LIN {X 0.160,Y -535.997,Z 395.131,A 0.000,B 0.000,C 90.000,E1 59.537} C_DIS
LIN {X 0.035,Y -538.957,Z 395.125,A 0.000,B 0.000,C 90.000,E1 58.408} C_DIS
LIN {X -0.234,Y -540.877,Z 395.120,A 0.000,B 0.000,C 90.000,E1 57.582} C_DIS
LIN {X -0.026,Y -542.349,Z 395.115,A 0.000,B 0.000,C 90.000,E1 56.707} C_DIS
LIN {X 0.021,Y -543.150,Z 395.112,A 0.000,B 0.000,C 90.000,E1 56.135} C_DIS
LIN {X -0.198,Y -544.070,Z 395.107,A 0.000,B 0.000,C 90.000,E1 55.308} C_DIS
LIN {X 0.313,Y -544.582,Z 395.104,A 0.000,B 0.000,C 90.000,E1 54.689} C_DIS
LIN {X 0.100,Y -544.932,Z 395.099,A 0.000,B 0.000,C 90.000,E1 53.863} C_DIS
LIN {X -0.151,Y -544.718,Z 395.091,A 0.000,B 0.000,C 90.000,E1 52.477} C_DIS
LIN {X -0.114,Y -544.668,Z 395.090,A 0.000,B 0.000,C 90.000,E1 52.190} C_DIS
LIN {X 0.024,Y -543.876,Z 395.084,A 0.000,B 0.000,C 90.000,E1 51.045} C_DIS
LIN {X 0.069,Y -542.657,Z 395.077,A 0.000,B 0.000,C 90.000,E1 49.908} C_DIS
LIN {X 0.102,Y -541.174,Z 395.071,A 0.000,B 0.000,C 90.000,E1 48.771} C_DIS
LIN {X -0.280,Y -539.163,Z 395.063,A 0.000,B 0.000,C 90.000,E1 47.391} C_DIS
LIN {X -0.056,Y -534.854,Z 395.047,A 0.000,B 0.000,C 90.000,E1 44.514} C_DIS
LIN {X 0.086,Y -531.734,Z 395.035,A 0.000,B 0.000,C 90.000,E1 42.204} C_DIS
LIN {X -0.062,Y -529.904,Z 395.027,A 0.000,B 0.000,C 90.000,E1 40.782} C_DIS
LIN {X -0.235,Y -528.110,Z 395.019,A 0.000,B 0.000,C 90.000,E1 39.358} C_DIS
LIN {X -0.060,Y -525.925,Z 395.009,A 0.000,B 0.000,C 90.000,E1 37.604} C_DIS
LIN {X 0.091,Y -524.030,Z 395.001,A 0.000,B 0.000,C 90.000,E1 36.137} C_DIS
LIN {X -0.034,Y -521.746,Z 394.991,A 0.000,B 0.000,C 90.000,E1 34.405} C_DIS
LIN {X -0.205,Y -519.458,Z 394.981,A 0.000,B 0.000,C 90.000,E1 32.673} C_DIS
LIN {X 0.171,Y -517.029,Z 394.972,A 0.000,B 0.000,C 90.000,E1 30.875} C_DIS
LIN {X 0.045,Y -514.873,Z 394.962,A 0.000,B 0.000,C 90.000,E1 29.127} C_DIS
LIN {X 0.264,Y -511.965,Z 394.949,A 0.000,B 0.000,C 90.000,E1 26.744} C_DIS
LIN {X -0.248,Y -510.001,Z 394.939,A 0.000,B 0.000,C 90.000,E1 25.027} C_DIS
LIN {X 0.226,Y -507.941,Z 394.927,A 0.000,B 0.000,C 90.000,E1 22.898} C_DIS
LIN {X -0.123,Y -506.318,Z 394.917,A 0.000,B 0.000,C 90.000,E1 21.153} C_DIS
LIN {X 0.245,Y -504.976,Z 394.908,A 0.000,B 0.000,C 90.000,E1 19.322} C_DIS
LIN {X -0.138,Y -503.539,Z 394.896,A 0.000,B 0.000,C 90.000,E1 17.275} C_DIS
LIN {X -0.210,Y -502.689,Z 394.888,A 0.000,B 0.000,C 90.000,E1 15.788} C_DIS
LIN {X 0.103,Y -501.504,Z 394.874,A 0.000,B 0.000,C 90.000,E1 13.355} C_DIS
LIN {X -0.150,Y -500.555,Z 394.854,A 0.000,B 0.000,C 90.000,E1 9.782} C_DIS
LIN {X 0.164,Y -500.484,Z 394.843,A 0.000,B 0.000,C 90.000,E1 7.644} C_DIS
LIN {X 0.217,Y -501.064,Z 394.828,A 0.000,B 0.000,C 90.000,E1 4.935} C_DIS
LIN {X -0.235,Y -503.237,Z 394.806,A 0.000,B 0.000,C 90.000,E1 1.088} C_DIS
LIN {X -0.242,Y -507.371,Z 394.784,A 0.000,B 0.000,C 90.000,E1 357.135} C_DIS
LIN {X 0.074,Y -510.722,Z 394.771,A 0.000,B 0.000,C 90.000,E1 354.723} C_DIS
LIN {X 0.122,Y -514.088,Z 394.759,A 0.000,B 0.000,C 90.000,E1 352.648} C_DIS
LIN {X -0.214,Y -519.053,Z 394.745,A 0.000,B 0.000,C 90.000,E1 350.038} C_DIS
LIN {X -0.215,Y -523.522,Z 394.733,A 0.000,B 0.000,C 90.000,E1 347.993} C_DIS
LIN {X 0.016,Y -528.565,Z 394.722,A 0.000,B 0.000,C 90.000,E1 345.936} C_DIS
LIN {X -0.045,Y -533.123,Z 394.712,A 0.000,B 0.000,C 90.000,E1 344.212} C_DIS
LIN {X -0.056,Y -536.981,Z 394.704,A 0.000,B 0.000,C 90.000,E1 342.779} C_DIS
LIN {X 0.217,Y -541.697,Z 394.695,A 0.000,B 0.000,C 90.000,E1 341.040} C_DIS
LIN {X -0.262,Y -546.551,Z 394.685,A 0.000,B 0.000,C 90.000,E1 339.390} C_DIS
LIN {X -0.168,Y -552.210,Z 394.674,A 0.000,B 0.000,C 90.000,E1 337.411} C_DIS
LIN {X -0.007,Y -556.377,Z 394.667,A 0.000,B 0.000,C 90.000,E1 335.997} C_DIS
LIN {X -0.126,Y -559.734,Z 394.661,A 0.000,B 0.000,C 90.000,E1 334.897} C_DIS
LIN {X 0.193,Y -564.865,Z 394.651,A 0.000,B 0.000,C 90.000,E1 333.204} C_DIS
LIN {X 0.030,Y -569.301,Z 394.644,A 0.000,B 0.000,C 90.000,E1 331.847} C_DIS
LIN {X -0.224,Y -571.851,Z 394.639,A 0.000,B 0.000,C 90.000,E1 331.051} C_DIS
LIN {X 0.218,Y -573.787,Z 394.636,A 0.000,B 0.000,C 90.000,E1 330.461} C_DIS
LIN {X -0.159,Y -579.145,Z 394.627,A 0.000,B 0.000,C 90.000,E1 328.869} C_DIS
LIN {X -0.149,Y -582.761,Z 394.621,A 0.000,B 0.000,C 90.000,E1 327.788} C_DIS
LIN {X -0.046,Y -588.119,Z 394.612,A 0.000,B 0.000,C 90.000,E1 326.167} C_DIS
LIN {X 0.135,Y -592.670,Z 394.605,A 0.000,B 0.000,C 90.000,E1 324.815} C_DIS
LIN {X 0.056,Y -597.283,Z 394.597,A 0.000,B 0.000,C 90.000,E1 323.497} C_DIS
LIN {X -0.047,Y -603.868,Z 394.587,A 0.000,B 0.000,C 90.000,E1 321.662} C_DIS
LIN {X 0.209,Y -609.580,Z 394.578,A 0.000,B 0.000,C 90.000,E1 320.070} C_DIS
LIN {X 0.210,Y -614.342,Z 394.571,A 0.000,B 0.000,C 90.000,E1 318.771} C_DIS
LIN {X 0.295,Y -619.034,Z 394.564,A 0.000,B 0.000,C 90.000,E1 317.472} C_DIS
LIN {X -0.001,Y -623.601,Z 394.557,A 0.000,B 0.000,C 90.000,E1 316.215} C_DIS
LIN {X 0.214,Y -628.170,Z 394.550,A 0.000,B 0.000,C 90.000,E1 314.919} C_DIS
LIN {X -0.147,Y -634.647,Z 394.540,A 0.000,B 0.000,C 90.000,E1 313.176} C_DIS
LIN {X -0.278,Y -640.243,Z 394.531,A 0.000,B 0.000,C 90.000,E1 311.676} C_DIS
LIN {X 0.334,Y -643.911,Z 394.526,A 0.000,B 0.000,C 90.000,E1 310.620} C_DIS
LIN {X 0.089,Y -647.469,Z 394.520,A 0.000,B 0.000,C 90.000,E1 309.644} C_DIS
LIN {X 0.323,Y -651.743,Z 394.513,A 0.000,B 0.000,C 90.000,E1 308.382} C_DIS
LIN {X 0.224,Y -655.835,Z 394.507,A 0.000,B 0.000,C 90.000,E1 307.156} C_DIS
LIN {X 0.187,Y -659.762,Z 394.500,A 0.000,B 0.000,C 90.000,E1 305.931} C_DIS
LIN {X -0.180,Y -663.485,Z 394.493,A 0.000,B 0.000,C 90.000,E1 304.739} C_DIS
LIN {X 0.194,Y -667.864,Z 394.485,A 0.000,B 0.000,C 90.000,E1 303.245} C_DIS
LIN {X -0.054,Y -671.506,Z 394.478,A 0.000,B 0.000,C 90.000,E1 302.054} C_DIS
LIN {X 0.016,Y -674.308,Z 394.473,A 0.000,B 0.000,C 90.000,E1 301.082} C_DIS
LIN {X -0.102,Y -676.921,Z 394.467,A 0.000,B 0.000,C 90.000,E1 300.129} C_DIS
LIN {X 0.057,Y -679.334,Z 394.462,A 0.000,B 0.000,C 90.000,E1 299.155} C_DIS
LIN {X -0.345,Y -681.547,Z 394.457,A 0.000,B 0.000,C 90.000,E1 298.231} C_DIS
LIN {X -0.333,Y -682.891,Z 394.453,A 0.000,B 0.000,C 90.000,E1 297.513} C_DIS
LIN {X -0.125,Y -683.417,Z 394.451,A 0.000,B 0.000,C 90.000,E1 297.257} C_DIS
LIN {X 0.031,Y -685.366,Z 394.445,A 0.000,B 0.000,C 90.000,E1 296.052} C_DIS
LIN {X 0.071,Y -686.370,Z 394.441,A 0.000,B 0.000,C 90.000,E1 295.335} C_DIS
LIN {X -0.176,Y -687.148,Z 394.437,A 0.000,B 0.000,C 90.000,E1 294.643} C_DIS
LIN {X -0.194,Y -687.808,Z 394.432,A 0.000,B 0.000,C 90.000,E1 293.695} C_DIS
LIN {X -0.245,Y -687.936,Z 394.430,A 0.000,B 0.000,C 90.000,E1 293.462} C_DIS
LIN {X -0.038,Y -687.795,Z 394.424,A 0.000,B 0.000,C 90.000,E1 292.259} C_DIS
LIN {X 0.102,Y -687.415,Z 394.420,A 0.000,B 0.000,C 90.000,E1 291.535} C_DIS
LIN {X 0.316,Y -687.210,Z 394.418,A 0.000,B 0.000,C 90.000,E1 291.280} C_DIS
LIN {X 0.281,Y -687.180,Z 394.417,A 0.000,B 0.000,C 90.000,E1 291.046} C_DIS
LIN {X -0.039,Y -686.081,Z 394.410,A 0.000,B 0.000,C 90.000,E1 289.885} C_DIS
LIN {X 0.268,Y -684.786,Z 394.404,A 0.000,B 0.000,C 90.000,E1 288.671} C_DIS
LIN {X -0.106,Y -683.115,Z 394.397,A 0.000,B 0.000,C 90.000,E1 287.511} C_DIS
LIN {X -0.138,Y -680.419,Z 394.388,A 0.000,B 0.000,C 90.000,E1 285.843} C_DIS
LIN {X -0.282,Y -678.802,Z 394.383,A 0.000,B 0.000,C 90.000,E1 284.898} C_DIS
LIN {X -0.011,Y -675.071,Z 394.371,A 0.000,B 0.000,C 90.000,E1 282.715} C_DIS
LIN {X -0.004,Y -671.647,Z 394.359,A 0.000,B 0.000,C 90.000,E1 280.546} C_DIS
LIN {X -0.157,Y -669.125,Z 394.348,A 0.000,B 0.000,C 90.000,E1 278.624} C_DIS
LIN {X -0.292,Y -666.348,Z 394.333,A 0.000,B 0.000,C 90.000,E1 275.967} C_DIS
LIN {X 0.307,Y -664.855,Z 394.321,A 0.000,B 0.000,C 90.000,E1 273.726} C_DIS
LIN {X 0.315,Y -663.862,Z 394.305,A 0.000,B 0.000,C 90.000,E1 270.802} C_DIS
LIN {X 0.131,Y -663.374,Z 394.298,A 0.000,B 0.000,C 90.000,E1 269.599} C_DIS
LIN {X -0.218,Y -662.840,Z 394.290,A 0.000,B 0.000,C 90.000,E1 268.165} C_DIS
LIN {X 0.232,Y -662.124,Z 394.283,A 0.000,B 0.000,C 90.000,E1 266.906} C_DIS
LIN {X -0.269,Y -661.643,Z 394.279,A 0.000,B 0.000,C 90.000,E1 266.216} C_DIS
LIN {X -0.111,Y -661.090,Z 394.275,A 0.000,B 0.000,C 90.000,E1 265.469} C_DIS
LIN {X 0.041,Y -660.205,Z 394.271,A 0.000,B 0.000,C 90.000,E1 264.723} C_DIS
LIN {X -0.279,Y -659.340,Z 394.268,A 0.000,B 0.000,C 90.000,E1 264.261} C_DIS
LIN {X 0.180,Y -659.100,Z 394.267,A 0.000,B 0.000,C 90.000,E1 263.976} C_DIS
LIN {X 0.052,Y -658.640,Z 394.265,A 0.000,B 0.000,C 90.000,E1 263.742} C_DIS
LIN {X 0.174,Y -657.627,Z 394.261,A 0.000,B 0.000,C 90.000,E1 262.996} C_DIS
LIN {X -0.288,Y -656.242,Z 394.257,A 0.000,B 0.000,C 90.000,E1 262.299} C_DIS
LIN {X -0.106,Y -654.761,Z 394.253,A 0.000,B 0.000,C 90.000,E1 261.546} C_DIS
LIN {X 0.208,Y -651.420,Z 394.245,A 0.000,B 0.000,C 90.000,E1 260.038} C_DIS
LIN {X -0.075,Y -647.533,Z 394.237,A 0.000,B 0.000,C 90.000,E1 258.578} C_DIS
LIN {X -0.285,Y -644.069,Z 394.230,A 0.000,B 0.000,C 90.000,E1 257.353} C_DIS
LIN {X 0.205,Y -640.363,Z 394.223,A 0.000,B 0.000,C 90.000,E1 256.061} C_DIS
LIN {X 0.168,Y -636.436,Z 394.216,A 0.000,B 0.000,C 90.000,E1 254.810} C_DIS
LIN {X -0.351,Y -633.973,Z 394.212,A 0.000,B 0.000,C 90.000,E1 254.102} C_DIS
LIN {X 0.103,Y -628.589,Z 394.203,A 0.000,B 0.000,C 90.000,E1 252.543} C_DIS
LIN {X 0.075,Y -624.788,Z 394.197,A 0.000,B 0.000,C 90.000,E1 251.529} C_DIS
LIN {X 0.190,Y -620.910,Z 394.192,A 0.000,B 0.000,C 90.000,E1 250.496} C_DIS
LIN {X 0.223,Y -615.912,Z 394.185,A 0.000,B 0.000,C 90.000,E1 249.209} C_DIS
LIN {X 0.171,Y -610.687,Z 394.177,A 0.000,B 0.000,C 90.000,E1 247.922} C_DIS
LIN {X 0.259,Y -605.253,Z 394.170,A 0.000,B 0.000,C 90.000,E1 246.613} C_DIS
LIN {X -0.294,Y -599.726,Z 394.163,A 0.000,B 0.000,C 90.000,E1 245.357} C_DIS
LIN {X -0.229,Y -593.037,Z 394.154,A 0.000,B 0.000,C 90.000,E1 243.768} C_DIS
LIN {X -0.037,Y -586.330,Z 394.145,A 0.000,B 0.000,C 90.000,E1 242.153} C_DIS
LIN {X 0.008,Y -579.744,Z 394.136,A 0.000,B 0.000,C 90.000,E1 240.539} C_DIS
LIN {X -0.217,Y -570.254,Z 394.123,A 0.000,B 0.000,C 90.000,E1 238.122} C_DIS
LIN {X 0.255,Y -562.350,Z 394.111,A 0.000,B 0.000,C 90.000,E1 235.881} C_DIS
LIN {X -0.195,Y -555.750,Z 394.100,A 0.000,B 0.000,C 90.000,E1 233.989} C_DIS
LIN {X 0.173,Y -551.060,Z 394.092,A 0.000,B 0.000,C 90.000,E1 232.557} C_DIS
LIN {X -0.030,Y -547.250,Z 394.086,A 0.000,B 0.000,C 90.000,E1 231.457} C_DIS
LIN {X 0.149,Y -540.560,Z 394.075,A 0.000,B 0.000,C 90.000,E1 229.461} C_DIS
LIN {X 0.097,Y -534.136,Z 394.064,A 0.000,B 0.000,C 90.000,E1 227.472} C_DIS
LIN {X 0.275,Y -528.807,Z 394.054,A 0.000,B 0.000,C 90.000,E1 225.729} C_DIS
LIN {X -0.169,Y -521.773,Z 394.041,A 0.000,B 0.000,C 90.000,E1 223.461} C_DIS
LIN {X 0.119,Y -516.634,Z 394.032,A 0.000,B 0.000,C 90.000,E1 221.676} C_DIS
LIN {X -0.219,Y -509.978,Z 394.019,A 0.000,B 0.000,C 90.000,E1 219.358} C_DIS
LIN {X -0.044,Y -506.009,Z 394.010,A 0.000,B 0.000,C 90.000,E1 217.855} C_DIS
LIN {X -0.278,Y -501.421,Z 394.000,A 0.000,B 0.000,C 90.000,E1 216.091} C_DIS
LIN {X -0.327,Y -496.158,Z 393.989,A 0.000,B 0.000,C 90.000,E1 213.992} C_DIS
LIN {X 0.044,Y -491.835,Z 393.979,A 0.000,B 0.000,C 90.000,E1 212.133} C_DIS
LIN {X 0.034,Y -486.888,Z 393.967,A 0.000,B 0.000,C 90.000,E1 210.001} C_DIS
LIN {X 0.071,Y -484.064,Z 393.960,A 0.000,B 0.000,C 90.000,E1 208.771} C_DIS
LIN {X -0.145,Y -480.517,Z 393.951,A 0.000,B 0.000,C 90.000,E1 207.257} C_DIS
LIN {X -0.227,Y -476.808,Z 393.943,A 0.000,B 0.000,C 90.000,E1 205.720} C_DIS
LIN {X 0.009,Y -472.373,Z 393.932,A 0.000,B 0.000,C 90.000,E1 203.823} C_DIS
LIN {X -0.106,Y -467.036,Z 393.920,A 0.000,B 0.000,C 90.000,E1 201.642} C_DIS
LIN {X 0.015,Y -460.484,Z 393.904,A 0.000,B 0.000,C 90.000,E1 198.779} C_DIS
LIN {X 0.059,Y -454.463,Z 393.888,A 0.000,B 0.000,C 90.000,E1 195.898} C_DIS
LIN {X 0.034,Y -450.183,Z 393.876,A 0.000,B 0.000,C 90.000,E1 193.647} C_DIS
LIN {X 0.131,Y -446.201,Z 393.863,A 0.000,B 0.000,C 90.000,E1 191.366} C_DIS
LIN {X -0.122,Y -443.009,Z 393.852,A 0.000,B 0.000,C 90.000,E1 189.443} C_DIS
LIN {X 0.072,Y -439.560,Z 393.840,A 0.000,B 0.000,C 90.000,E1 187.125} C_DIS
LIN {X -0.022,Y -435.320,Z 393.821,A 0.000,B 0.000,C 90.000,E1 183.841} C_DIS
LIN {X -0.044,Y -432.260,Z 393.805,A 0.000,B 0.000,C 90.000,E1 180.859} C_DIS
LIN {X -0.094,Y -430.054,Z 393.786,A 0.000,B 0.000,C 90.000,E1 177.535} C_DIS
LIN {X -0.163,Y -428.872,Z 393.768,A 0.000,B 0.000,C 90.000,E1 174.204} C_DIS
LIN {X 0.128,Y -428.887,Z 393.745,A 0.000,B 0.000,C 90.000,E1 170.151} C_DIS
LIN {X 0.211,Y -431.011,Z 393.719,A 0.000,B 0.000,C 90.000,E1 165.463} C_DIS
LIN {X 0.097,Y -434.226,Z 393.699,A 0.000,B 0.000,C 90.000,E1 161.819} C_DIS
LIN {X -0.128,Y -438.181,Z 393.681,A 0.000,B 0.000,C 90.000,E1 158.539} C_DIS
LIN {X 0.198,Y -442.586,Z 393.664,A 0.000,B 0.000,C 90.000,E1 155.537} C_DIS
LIN {X 0.012,Y -447.200,Z 393.650,A 0.000,B 0.000,C 90.000,E1 152.948} C_DIS
LIN {X -0.163,Y -454.671,Z 393.630,A 0.000,B 0.000,C 90.000,E1 149.410} C_DIS
LIN {X 0.054,Y -464.558,Z 393.609,A 0.000,B 0.000,C 90.000,E1 145.548} C_DIS
LIN {X -0.005,Y -473.109,Z 393.593,A 0.000,B 0.000,C 90.000,E1 142.718} C_DIS
LIN {X 0.157,Y -480.287,Z 393.581,A 0.000,B 0.000,C 90.000,E1 140.517} C_DIS
LIN {X -0.183,Y -485.401,Z 393.572,A 0.000,B 0.000,C 90.000,E1 139.013} C_DIS
LIN {X 0.066,Y -489.486,Z 393.565,A 0.000,B 0.000,C 90.000,E1 137.757} C_DIS
LIN {X 0.049,Y -493.261,Z 393.559,A 0.000,B 0.000,C 90.000,E1 136.539} C_DIS
LIN {X 0.067,Y -496.812,Z 393.552,A 0.000,B 0.000,C 90.000,E1 135.324} C_DIS
LIN {X 0.142,Y -500.146,Z 393.545,A 0.000,B 0.000,C 90.000,E1 134.109} C_DIS
LIN {X -0.085,Y -503.015,Z 393.539,A 0.000,B 0.000,C 90.000,E1 132.933} C_DIS
LIN {X 0.224,Y -504.898,Z 393.534,A 0.000,B 0.000,C 90.000,E1 132.000} C_DIS
LIN {X -0.162,Y -506.549,Z 393.529,A 0.000,B 0.000,C 90.000,E1 131.148} C_DIS
LIN {X -0.046,Y -507.556,Z 393.525,A 0.000,B 0.000,C 90.000,E1 130.539} C_DIS
LIN {X -0.021,Y -508.812,Z 393.520,A 0.000,B 0.000,C 90.000,E1 129.644} C_DIS
LIN {X 0.017,Y -509.652,Z 393.515,A 0.000,B 0.000,C 90.000,E1 128.749} C_DIS
LIN {X -0.254,Y -510.040,Z 393.510,A 0.000,B 0.000,C 90.000,E1 127.890} C_DIS
LIN {X -0.119,Y -509.884,Z 393.507,A 0.000,B 0.000,C 90.000,E1 127.282} C_DIS
LIN {X 0.110,Y -509.562,Z 393.504,A 0.000,B 0.000,C 90.000,E1 126.664} C_DIS
LIN {X -0.158,Y -508.689,Z 393.499,A 0.000,B 0.000,C 90.000,E1 125.804} C_DIS
LIN {X -0.023,Y -507.448,Z 393.494,A 0.000,B 0.000,C 90.000,E1 124.898} C_DIS
LIN {X 0.099,Y -505.939,Z 393.489,A 0.000,B 0.000,C 90.000,E1 123.992} C_DIS
LIN {X -0.112,Y -504.696,Z 393.486,A 0.000,B 0.000,C 90.000,E1 123.420} C_DIS
LIN {X -0.187,Y -503.259,Z 393.482,A 0.000,B 0.000,C 90.000,E1 122.832} C_DIS
LIN {X 0.177,Y -499.714,Z 393.476,A 0.000,B 0.000,C 90.000,E1 121.592} C_DIS
LIN {X 0.076,Y -497.729,Z 393.472,A 0.000,B 0.000,C 90.000,E1 121.003} C_DIS
LIN {X -0.036,Y -495.545,Z 393.469,A 0.000,B 0.000,C 90.000,E1 120.413} C_DIS
LIN {X 0.109,Y -492.140,Z 393.464,A 0.000,B 0.000,C 90.000,E1 119.489} C_DIS
LIN {X -0.219,Y -488.355,Z 393.459,A 0.000,B 0.000,C 90.000,E1 118.615} C_DIS
LIN {X -0.174,Y -482.956,Z 393.452,A 0.000,B 0.000,C 90.000,E1 117.385} C_DIS
LIN {X -0.012,Y -476.366,Z 393.444,A 0.000,B 0.000,C 90.000,E1 115.976} C_DIS
LIN {X -0.125,Y -471.103,Z 393.438,A 0.000,B 0.000,C 90.000,E1 114.899} C_DIS
LIN {X -0.125,Y -464.828,Z 393.431,A 0.000,B 0.000,C 90.000,E1 113.643} C_DIS
LIN {X -0.144,Y -460.146,Z 393.426,A 0.000,B 0.000,C 90.000,E1 112.695} C_DIS
LIN {X -0.051,Y -453.275,Z 393.418,A 0.000,B 0.000,C 90.000,E1 111.280} C_DIS
LIN {X -0.091,Y -453.268,Z 393.418,A 0.000,B 0.000,C 90.000,E1 111.280} C_DIS
LIN {X -0.158,Y -457.292,Z 393.410,A 0.000,B 0.000,C 90.000,E1 109.812} C_DIS
LIN {X -0.090,Y -465.913,Z 393.387,A 0.000,B 0.000,C 90.000,E1 105.662} C_DIS
LIN {X 0.081,Y -467.476,Z 393.383,A 0.000,B 0.000,C 90.000,E1 105.009} C_DIS
LIN {X -0.114,Y -468.076,Z 393.382,A 0.000,B 0.000,C 90.000,E1 104.717} C_DIS
LIN {X 0.025,Y -475.726,Z 393.357,A 0.000,B 0.000,C 90.000,E1 100.310} C_DIS
LIN {X -0.138,Y -476.272,Z 393.356,A 0.000,B 0.000,C 90.000,E1 100.018} C_DIS
LIN {X 0.127,Y -482.156,Z 393.330,A 0.000,B 0.000,C 90.000,E1 95.334} C_DIS
LIN {X -0.119,Y -485.537,Z 393.304,A 0.000,B 0.000,C 90.000,E1 90.745} C_DIS
LIN {X 0.089,Y -486.301,Z 393.282,A 0.000,B 0.000,C 90.000,E1 86.731} C_DIS
LIN {X 0.223,Y -486.330,Z 393.279,A 0.000,B 0.000,C 90.000,E1 86.102} C_DIS
LIN {X -0.184,Y -484.637,Z 393.253,A 0.000,B 0.000,C 90.000,E1 81.546} C_DIS
LIN {X 0.175,Y -480.562,Z 393.227,A 0.000,B 0.000,C 90.000,E1 76.881} C_DIS
LIN {X 0.085,Y -474.321,Z 393.201,A 0.000,B 0.000,C 90.000,E1 72.236} C_DIS
LIN {X -0.093,Y -473.923,Z 393.200,A 0.000,B 0.000,C 90.000,E1 71.945} C_DIS
LIN {X 0.094,Y -471.898,Z 393.194,A 0.000,B 0.000,C 90.000,E1 70.913} C_DIS
LIN {X 0.055,Y -471.896,Z 393.194,A 0.000,B 0.000,C 90.000,E1 70.913} C_DIS
LIN {X -0.036,Y -482.726,Z 393.186,A 0.000,B 0.000,C 90.000,E1 69.444} C_DIS
LIN {X -0.166,Y -491.817,Z 393.179,A 0.000,B 0.000,C 90.000,E1 68.230} C_DIS
LIN {X -0.245,Y -499.391,Z 393.173,A 0.000,B 0.000,C 90.000,E1 67.177} C_DIS
LIN {X -0.027,Y -506.588,Z 393.167,A 0.000,B 0.000,C 90.000,E1 66.102} C_DIS
LIN {X -0.021,Y -511.308,Z 393.163,A 0.000,B 0.000,C 90.000,E1 65.357} C_DIS
LIN {X 0.243,Y -515.701,Z 393.159,A 0.000,B 0.000,C 90.000,E1 64.588} C_DIS
LIN {X 0.027,Y -518.913,Z 393.156,A 0.000,B 0.000,C 90.000,E1 64.024} C_DIS
LIN {X 0.207,Y -523.160,Z 393.151,A 0.000,B 0.000,C 90.000,E1 63.127} C_DIS
LIN {X -0.034,Y -527.156,Z 393.146,A 0.000,B 0.000,C 90.000,E1 62.281} C_DIS
LIN {X 0.230,Y -530.468,Z 393.141,A 0.000,B 0.000,C 90.000,E1 61.385} C_DIS
LIN {X -0.112,Y -532.522,Z 393.138,A 0.000,B 0.000,C 90.000,E1 60.845} C_DIS
LIN {X -0.261,Y -535.158,Z 393.133,A 0.000,B 0.000,C 90.000,E1 59.999} C_DIS
LIN {X -0.105,Y -536.809,Z 393.130,A 0.000,B 0.000,C 90.000,E1 59.410} C_DIS
LIN {X 0.062,Y -539.735,Z 393.124,A 0.000,B 0.000,C 90.000,E1 58.250} C_DIS
LIN {X 0.263,Y -541.580,Z 393.119,A 0.000,B 0.000,C 90.000,E1 57.375} C_DIS
LIN {X 0.028,Y -543.044,Z 393.114,A 0.000,B 0.000,C 90.000,E1 56.548} C_DIS
LIN {X -0.221,Y -543.860,Z 393.111,A 0.000,B 0.000,C 90.000,E1 56.008} C_DIS
LIN {X 0.012,Y -544.812,Z 393.106,A 0.000,B 0.000,C 90.000,E1 55.135} C_DIS
LIN {X 0.080,Y -545.357,Z 393.103,A 0.000,B 0.000,C 90.000,E1 54.562} C_DIS
LIN {X 0.194,Y -545.722,Z 393.099,A 0.000,B 0.000,C 90.000,E1 53.703} C_DIS
LIN {X -0.038,Y -545.505,Z 393.091,A 0.000,B 0.000,C 90.000,E1 52.316} C_DIS
LIN {X 0.043,Y -545.274,Z 393.088,A 0.000,B 0.000,C 90.000,E1 51.743} C_DIS
LIN {X 0.120,Y -544.925,Z 393.084,A 0.000,B 0.000,C 90.000,E1 51.170} C_DIS
LIN {X -0.165,Y -543.780,Z 393.078,A 0.000,B 0.000,C 90.000,E1 50.070} C_DIS
LIN {X -0.117,Y -542.392,Z 393.072,A 0.000,B 0.000,C 90.000,E1 48.933} C_DIS
LIN {X 0.282,Y -540.399,Z 393.064,A 0.000,B 0.000,C 90.000,E1 47.472} C_DIS
LIN {X -0.175,Y -536.898,Z 393.051,A 0.000,B 0.000,C 90.000,E1 45.243} C_DIS
LIN {X 0.088,Y -534.453,Z 393.042,A 0.000,B 0.000,C 90.000,E1 43.500} C_DIS
LIN {X -0.121,Y -531.835,Z 393.031,A 0.000,B 0.000,C 90.000,E1 41.515} C_DIS
LIN {X 0.034,Y -529.309,Z 393.019,A 0.000,B 0.000,C 90.000,E1 39.483} C_DIS
LIN {X 0.199,Y -526.745,Z 393.008,A 0.000,B 0.000,C 90.000,E1 37.443} C_DIS
LIN {X 0.015,Y -524.459,Z 392.999,A 0.000,B 0.000,C 90.000,E1 35.724} C_DIS
LIN {X -0.096,Y -522.158,Z 392.989,A 0.000,B 0.000,C 90.000,E1 33.992} C_DIS
LIN {X -0.201,Y -520.230,Z 392.981,A 0.000,B 0.000,C 90.000,E1 32.546} C_DIS
LIN {X 0.089,Y -518.265,Z 392.973,A 0.000,B 0.000,C 90.000,E1 31.052} C_DIS
LIN {X 0.090,Y -515.692,Z 392.961,A 0.000,B 0.000,C 90.000,E1 28.999} C_DIS
LIN {X -0.009,Y -513.169,Z 392.950,A 0.000,B 0.000,C 90.000,E1 26.950} C_DIS
LIN {X 0.194,Y -511.214,Z 392.940,A 0.000,B 0.000,C 90.000,E1 25.155} C_DIS
LIN {X -0.133,Y -508.859,Z 392.927,A 0.000,B 0.000,C 90.000,E1 22.823} C_DIS
LIN {X -0.179,Y -507.241,Z 392.917,A 0.000,B 0.000,C 90.000,E1 21.046} C_DIS
LIN {X -0.255,Y -505.920,Z 392.907,A 0.000,B 0.000,C 90.000,E1 19.268} C_DIS
LIN {X 0.024,Y -504.500,Z 392.895,A 0.000,B 0.000,C 90.000,E1 17.149} C_DIS
LIN {X -0.037,Y -503.665,Z 392.887,A 0.000,B 0.000,C 90.000,E1 15.662} C_DIS
LIN {X 0.181,Y -502.554,Z 392.874,A 0.000,B 0.000,C 90.000,E1 13.244} C_DIS
LIN {X -0.012,Y -501.654,Z 392.854,A 0.000,B 0.000,C 90.000,E1 9.670} C_DIS
LIN {X -0.018,Y -501.620,Z 392.844,A 0.000,B 0.000,C 90.000,E1 7.871} C_DIS
LIN {X 0.062,Y -502.191,Z 392.829,A 0.000,B 0.000,C 90.000,E1 5.163} C_DIS
LIN {X 0.160,Y -504.312,Z 392.807,A 0.000,B 0.000,C 90.000,E1 1.260} C_DIS
LIN {X -0.199,Y -508.685,Z 392.784,A 0.000,B 0.000,C 90.000,E1 357.135} C_DIS
LIN {X -0.016,Y -510.229,Z 392.777,A 0.000,B 0.000,C 90.000,E1 355.927} C_DIS
LIN {X 0.156,Y -512.034,Z 392.771,A 0.000,B 0.000,C 90.000,E1 354.723} C_DIS
LIN {X 0.239,Y -515.444,Z 392.759,A 0.000,B 0.000,C 90.000,E1 352.648} C_DIS
LIN {X -0.050,Y -520.452,Z 392.745,A 0.000,B 0.000,C 90.000,E1 350.038} C_DIS
LIN {X 0.079,Y -528.533,Z 392.725,A 0.000,B 0.000,C 90.000,E1 346.533} C_DIS
LIN {X 0.230,Y -534.599,Z 392.712,A 0.000,B 0.000,C 90.000,E1 344.212} C_DIS
LIN {X 0.248,Y -538.483,Z 392.705,A 0.000,B 0.000,C 90.000,E1 342.779} C_DIS
LIN {X 0.043,Y -543.218,Z 392.695,A 0.000,B 0.000,C 90.000,E1 341.094} C_DIS
LIN {X 0.112,Y -548.063,Z 392.686,A 0.000,B 0.000,C 90.000,E1 339.390} C_DIS
LIN {X 0.250,Y -553.769,Z 392.675,A 0.000,B 0.000,C 90.000,E1 337.411} C_DIS
LIN {X -0.068,Y -557.924,Z 392.667,A 0.000,B 0.000,C 90.000,E1 336.049} C_DIS
LIN {X 0.109,Y -561.298,Z 392.661,A 0.000,B 0.000,C 90.000,E1 334.921} C_DIS
LIN {X -0.168,Y -568.151,Z 392.649,A 0.000,B 0.000,C 90.000,E1 332.743} C_DIS
LIN {X 0.069,Y -570.768,Z 392.644,A 0.000,B 0.000,C 90.000,E1 331.897} C_DIS
LIN {X 0.131,Y -576.207,Z 392.635,A 0.000,B 0.000,C 90.000,E1 330.255} C_DIS
LIN {X -0.193,Y -581.578,Z 392.626,A 0.000,B 0.000,C 90.000,E1 328.663} C_DIS
LIN {X -0.148,Y -585.178,Z 392.620,A 0.000,B 0.000,C 90.000,E1 327.582} C_DIS
LIN {X -0.074,Y -592.409,Z 392.608,A 0.000,B 0.000,C 90.000,E1 325.435} C_DIS
LIN {X 0.078,Y -597.899,Z 392.599,A 0.000,B 0.000,C 90.000,E1 323.829} C_DIS
LIN {X 0.104,Y -604.488,Z 392.589,A 0.000,B 0.000,C 90.000,E1 321.984} C_DIS
LIN {X 0.172,Y -611.144,Z 392.579,A 0.000,B 0.000,C 90.000,E1 320.150} C_DIS
LIN {X 0.198,Y -615.929,Z 392.572,A 0.000,B 0.000,C 90.000,E1 318.852} C_DIS
LIN {X 0.309,Y -620.621,Z 392.564,A 0.000,B 0.000,C 90.000,E1 317.553} C_DIS
LIN {X 0.039,Y -625.199,Z 392.557,A 0.000,B 0.000,C 90.000,E1 316.296} C_DIS
LIN {X 0.281,Y -629.771,Z 392.550,A 0.000,B 0.000,C 90.000,E1 315.000} C_DIS
LIN {X 0.061,Y -635.300,Z 392.542,A 0.000,B 0.000,C 90.000,E1 313.500} C_DIS
LIN {X -0.050,Y -640.885,Z 392.533,A 0.000,B 0.000,C 90.000,E1 312.000} C_DIS
LIN {X 0.008,Y -645.481,Z 392.526,A 0.000,B 0.000,C 90.000,E1 310.744} C_DIS
LIN {X 0.274,Y -649.049,Z 392.521,A 0.000,B 0.000,C 90.000,E1 309.725} C_DIS
LIN {X -0.379,Y -653.332,Z 392.514,A 0.000,B 0.000,C 90.000,E1 308.543} C_DIS
LIN {X -0.054,Y -657.427,Z 392.507,A 0.000,B 0.000,C 90.000,E1 307.282} C_DIS
LIN {X -0.461,Y -661.379,Z 392.500,A 0.000,B 0.000,C 90.000,E1 306.091} C_DIS
LIN {X -0.304,Y -665.870,Z 392.492,A 0.000,B 0.000,C 90.000,E1 304.612} C_DIS
LIN {X -0.437,Y -670.207,Z 392.484,A 0.000,B 0.000,C 90.000,E1 303.166} C_DIS
LIN {X -0.086,Y -673.807,Z 392.477,A 0.000,B 0.000,C 90.000,E1 301.926} C_DIS
LIN {X -0.158,Y -675.860,Z 392.473,A 0.000,B 0.000,C 90.000,E1 301.209} C_DIS
LIN {X -0.071,Y -679.108,Z 392.467,A 0.000,B 0.000,C 90.000,E1 300.001} C_DIS
LIN {X -0.081,Y -680.904,Z 392.463,A 0.000,B 0.000,C 90.000,E1 299.283} C_DIS
LIN {X 0.137,Y -683.010,Z 392.457,A 0.000,B 0.000,C 90.000,E1 298.309} C_DIS
LIN {X -0.225,Y -684.745,Z 392.452,A 0.000,B 0.000,C 90.000,E1 297.385} C_DIS
LIN {X 0.172,Y -686.802,Z 392.444,A 0.000,B 0.000,C 90.000,E1 295.924} C_DIS
LIN {X 0.002,Y -687.398,Z 392.442,A 0.000,B 0.000,C 90.000,E1 295.463} C_DIS
LIN {X -0.236,Y -688.034,Z 392.438,A 0.000,B 0.000,C 90.000,E1 294.771} C_DIS
LIN {X -0.016,Y -688.671,Z 392.431,A 0.000,B 0.000,C 90.000,E1 293.567} C_DIS
LIN {X 0.119,Y -688.667,Z 392.427,A 0.000,B 0.000,C 90.000,E1 292.845} C_DIS
LIN {X -0.106,Y -688.398,Z 392.423,A 0.000,B 0.000,C 90.000,E1 292.153} C_DIS
LIN {X -0.378,Y -687.677,Z 392.418,A 0.000,B 0.000,C 90.000,E1 291.227} C_DIS
LIN {X 0.187,Y -686.316,Z 392.411,A 0.000,B 0.000,C 90.000,E1 289.993} C_DIS
LIN {X 0.128,Y -685.554,Z 392.409,A 0.000,B 0.000,C 90.000,E1 289.523} C_DIS
LIN {X 0.326,Y -685.334,Z 392.407,A 0.000,B 0.000,C 90.000,E1 289.268} C_DIS
LIN {X -0.160,Y -684.724,Z 392.405,A 0.000,B 0.000,C 90.000,E1 288.833} C_DIS
LIN {X -0.102,Y -682.888,Z 392.398,A 0.000,B 0.000,C 90.000,E1 287.638} C_DIS
LIN {X 0.015,Y -679.678,Z 392.387,A 0.000,B 0.000,C 90.000,E1 285.717} C_DIS
LIN {X -0.143,Y -677.976,Z 392.382,A 0.000,B 0.000,C 90.000,E1 284.773} C_DIS
LIN {X 0.143,Y -674.623,Z 392.371,A 0.000,B 0.000,C 90.000,E1 282.827} C_DIS
LIN {X -0.065,Y -670.735,Z 392.358,A 0.000,B 0.000,C 90.000,E1 280.433} C_DIS
LIN {X -0.151,Y -668.513,Z 392.349,A 0.000,B 0.000,C 90.000,E1 278.746} C_DIS
LIN {X -0.107,Y -665.910,Z 392.335,A 0.000,B 0.000,C 90.000,E1 276.315} C_DIS
LIN {X -0.303,Y -664.207,Z 392.322,A 0.000,B 0.000,C 90.000,E1 273.898} C_DIS
LIN {X -0.153,Y -663.265,Z 392.307,A 0.000,B 0.000,C 90.000,E1 271.203} C_DIS
LIN {X 0.167,Y -663.194,Z 392.304,A 0.000,B 0.000,C 90.000,E1 270.688} C_DIS
LIN {X -0.027,Y -662.700,Z 392.297,A 0.000,B 0.000,C 90.000,E1 269.484} C_DIS
LIN {X -0.235,Y -662.339,Z 392.290,A 0.000,B 0.000,C 90.000,E1 268.282} C_DIS
LIN {X 0.229,Y -661.739,Z 392.284,A 0.000,B 0.000,C 90.000,E1 267.020} C_DIS
LIN {X 0.203,Y -661.303,Z 392.278,A 0.000,B 0.000,C 90.000,E1 266.045} C_DIS
LIN {X -0.303,Y -660.972,Z 392.274,A 0.000,B 0.000,C 90.000,E1 265.355} C_DIS
LIN {X -0.154,Y -660.239,Z 392.270,A 0.000,B 0.000,C 90.000,E1 264.609} C_DIS
LIN {X -0.267,Y -658.734,Z 392.263,A 0.000,B 0.000,C 90.000,E1 263.394} C_DIS
LIN {X -0.145,Y -657.587,Z 392.259,A 0.000,B 0.000,C 90.000,E1 262.648} C_DIS
LIN {X -0.075,Y -655.745,Z 392.254,A 0.000,B 0.000,C 90.000,E1 261.659} C_DIS
LIN {X 0.103,Y -654.122,Z 392.250,A 0.000,B 0.000,C 90.000,E1 260.905} C_DIS
LIN {X 0.024,Y -651.875,Z 392.244,A 0.000,B 0.000,C 90.000,E1 259.926} C_DIS
LIN {X 0.142,Y -649.432,Z 392.239,A 0.000,B 0.000,C 90.000,E1 258.926} C_DIS
LIN {X 0.244,Y -647.576,Z 392.234,A 0.000,B 0.000,C 90.000,E1 258.173} C_DIS
LIN {X 0.169,Y -644.210,Z 392.228,A 0.000,B 0.000,C 90.000,E1 256.937} C_DIS
LIN {X 0.041,Y -640.537,Z 392.221,A 0.000,B 0.000,C 90.000,E1 255.700} C_DIS
LIN {X 0.015,Y -636.610,Z 392.214,A 0.000,B 0.000,C 90.000,E1 254.448} C_DIS
LIN {X -0.073,Y -632.279,Z 392.207,A 0.000,B 0.000,C 90.000,E1 253.196} C_DIS
LIN {X -0.041,Y -628.653,Z 392.201,A 0.000,B 0.000,C 90.000,E1 252.181} C_DIS
LIN {X -0.080,Y -623.930,Z 392.194,A 0.000,B 0.000,C 90.000,E1 250.913} C_DIS
LIN {X -0.226,Y -617.912,Z 392.185,A 0.000,B 0.000,C 90.000,E1 249.390} C_DIS
LIN {X -0.238,Y -612.734,Z 392.178,A 0.000,B 0.000,C 90.000,E1 248.103} C_DIS
LIN {X -0.110,Y -607.337,Z 392.171,A 0.000,B 0.000,C 90.000,E1 246.794} C_DIS
LIN {X -0.074,Y -601.812,Z 392.164,A 0.000,B 0.000,C 90.000,E1 245.485} C_DIS
LIN {X 0.112,Y -596.276,Z 392.157,A 0.000,B 0.000,C 90.000,E1 244.152} C_DIS
LIN {X 0.096,Y -589.576,Z 392.148,A 0.000,B 0.000,C 90.000,E1 242.564} C_DIS
LIN {X -0.029,Y -582.948,Z 392.139,A 0.000,B 0.000,C 90.000,E1 240.973} C_DIS
LIN {X 0.215,Y -574.392,Z 392.127,A 0.000,B 0.000,C 90.000,E1 238.791} C_DIS
LIN {X 0.139,Y -565.374,Z 392.113,A 0.000,B 0.000,C 90.000,E1 236.342} C_DIS
LIN {X -0.006,Y -557.826,Z 392.101,A 0.000,B 0.000,C 90.000,E1 234.149} C_DIS
LIN {X -0.123,Y -554.106,Z 392.095,A 0.000,B 0.000,C 90.000,E1 233.050} C_DIS
LIN {X 0.155,Y -550.314,Z 392.089,A 0.000,B 0.000,C 90.000,E1 231.904} C_DIS
LIN {X 0.024,Y -544.555,Z 392.079,A 0.000,B 0.000,C 90.000,E1 230.231} C_DIS
LIN {X -0.313,Y -539.847,Z 392.071,A 0.000,B 0.000,C 90.000,E1 228.852} C_DIS
LIN {X 0.023,Y -534.390,Z 392.062,A 0.000,B 0.000,C 90.000,E1 227.106} C_DIS
LIN {X 0.238,Y -529.976,Z 392.054,A 0.000,B 0.000,C 90.000,E1 225.648} C_DIS
LIN {X -0.175,Y -522.912,Z 392.041,A 0.000,B 0.000,C 90.000,E1 223.380} C_DIS
LIN {X 0.139,Y -517.780,Z 392.031,A 0.000,B 0.000,C 90.000,E1 221.595} C_DIS
LIN {X -0.168,Y -511.128,Z 392.018,A 0.000,B 0.000,C 90.000,E1 219.277} C_DIS
LIN {X -0.287,Y -507.130,Z 392.010,A 0.000,B 0.000,C 90.000,E1 217.810} C_DIS
LIN {X 0.106,Y -501.762,Z 391.998,A 0.000,B 0.000,C 90.000,E1 215.678} C_DIS
LIN {X 0.065,Y -496.517,Z 391.987,A 0.000,B 0.000,C 90.000,E1 213.579} C_DIS
LIN {X -0.086,Y -492.955,Z 391.978,A 0.000,B 0.000,C 90.000,E1 212.084} C_DIS
LIN {X -0.056,Y -488.708,Z 391.968,A 0.000,B 0.000,C 90.000,E1 210.256} C_DIS
LIN {X -0.188,Y -485.188,Z 391.960,A 0.000,B 0.000,C 90.000,E1 208.743} C_DIS
LIN {X -0.178,Y -482.386,Z 391.953,A 0.000,B 0.000,C 90.000,E1 207.513} C_DIS
LIN {X -0.225,Y -478.717,Z 391.944,A 0.000,B 0.000,C 90.000,E1 205.976} C_DIS
LIN {X 0.058,Y -474.290,Z 391.934,A 0.000,B 0.000,C 90.000,E1 204.079} C_DIS
LIN {X 0.083,Y -470.453,Z 391.925,A 0.000,B 0.000,C 90.000,E1 202.514} C_DIS
LIN {X -0.148,Y -466.728,Z 391.916,A 0.000,B 0.000,C 90.000,E1 200.972} C_DIS
LIN {X 0.045,Y -460.955,Z 391.902,A 0.000,B 0.000,C 90.000,E1 198.417} C_DIS
LIN {X -0.120,Y -456.304,Z 391.890,A 0.000,B 0.000,C 90.000,E1 196.205} C_DIS
LIN {X 0.223,Y -451.375,Z 391.876,A 0.000,B 0.000,C 90.000,E1 193.592} C_DIS
LIN {X -0.083,Y -447.355,Z 391.863,A 0.000,B 0.000,C 90.000,E1 191.366} C_DIS
LIN {X 0.201,Y -444.139,Z 391.852,A 0.000,B 0.000,C 90.000,E1 189.378} C_DIS
LIN {X -0.083,Y -440.677,Z 391.840,A 0.000,B 0.000,C 90.000,E1 187.125} C_DIS
LIN {X -0.132,Y -436.396,Z 391.821,A 0.000,B 0.000,C 90.000,E1 183.841} C_DIS
LIN {X -0.026,Y -433.049,Z 391.803,A 0.000,B 0.000,C 90.000,E1 180.516} C_DIS
LIN {X -0.047,Y -430.932,Z 391.784,A 0.000,B 0.000,C 90.000,E1 177.192} C_DIS
LIN {X -0.045,Y -429.838,Z 391.766,A 0.000,B 0.000,C 90.000,E1 173.856} C_DIS
LIN {X 0.096,Y -430.114,Z 391.740,A 0.000,B 0.000,C 90.000,E1 169.162} C_DIS
LIN {X -0.185,Y -432.441,Z 391.716,A 0.000,B 0.000,C 90.000,E1 164.866} C_DIS
LIN {X -0.160,Y -435.159,Z 391.699,A 0.000,B 0.000,C 90.000,E1 161.873} C_DIS
LIN {X -0.180,Y -438.703,Z 391.683,A 0.000,B 0.000,C 90.000,E1 158.901} C_DIS
LIN {X 0.137,Y -444.635,Z 391.661,A 0.000,B 0.000,C 90.000,E1 154.921} C_DIS
LIN {X -0.194,Y -449.401,Z 391.646,A 0.000,B 0.000,C 90.000,E1 152.359} C_DIS
LIN {X -0.036,Y -457.157,Z 391.627,A 0.000,B 0.000,C 90.000,E1 148.791} C_DIS
LIN {X 0.150,Y -463.763,Z 391.612,A 0.000,B 0.000,C 90.000,E1 146.215} C_DIS
LIN {X -0.199,Y -472.185,Z 391.597,A 0.000,B 0.000,C 90.000,E1 143.417} C_DIS
LIN {X -0.056,Y -479.266,Z 391.585,A 0.000,B 0.000,C 90.000,E1 141.215} C_DIS
LIN {X -0.158,Y -483.393,Z 391.578,A 0.000,B 0.000,C 90.000,E1 139.989} C_DIS
LIN {X -0.266,Y -487.503,Z 391.571,A 0.000,B 0.000,C 90.000,E1 138.771} C_DIS
LIN {X 0.020,Y -491.549,Z 391.564,A 0.000,B 0.000,C 90.000,E1 137.514} C_DIS
LIN {X 0.034,Y -495.288,Z 391.557,A 0.000,B 0.000,C 90.000,E1 136.296} C_DIS
LIN {X 0.084,Y -498.797,Z 391.551,A 0.000,B 0.000,C 90.000,E1 135.081} C_DIS
LIN {X -0.020,Y -501.294,Z 391.546,A 0.000,B 0.000,C 90.000,E1 134.190} C_DIS
LIN {X -0.230,Y -504.159,Z 391.539,A 0.000,B 0.000,C 90.000,E1 133.014} C_DIS
LIN {X 0.316,Y -506.661,Z 391.532,A 0.000,B 0.000,C 90.000,E1 131.757} C_DIS
LIN {X -0.156,Y -508.749,Z 391.526,A 0.000,B 0.000,C 90.000,E1 130.620} C_DIS
LIN {X -0.116,Y -509.996,Z 391.521,A 0.000,B 0.000,C 90.000,E1 129.725} C_DIS
LIN {X -0.065,Y -510.868,Z 391.516,A 0.000,B 0.000,C 90.000,E1 128.830} C_DIS
LIN {X 0.079,Y -511.234,Z 391.512,A 0.000,B 0.000,C 90.000,E1 128.222} C_DIS
LIN {X -0.092,Y -511.306,Z 391.509,A 0.000,B 0.000,C 90.000,E1 127.649} C_DIS
LIN {X 0.066,Y -510.914,Z 391.504,A 0.000,B 0.000,C 90.000,E1 126.744} C_DIS
LIN {X -0.187,Y -510.121,Z 391.499,A 0.000,B 0.000,C 90.000,E1 125.884} C_DIS
LIN {X -0.034,Y -508.970,Z 391.494,A 0.000,B 0.000,C 90.000,E1 124.978} C_DIS
LIN {X 0.107,Y -507.491,Z 391.489,A 0.000,B 0.000,C 90.000,E1 124.072} C_DIS
LIN {X -0.092,Y -506.279,Z 391.486,A 0.000,B 0.000,C 90.000,E1 123.499} C_DIS
LIN {X -0.262,Y -504.049,Z 391.481,A 0.000,B 0.000,C 90.000,E1 122.625} C_DIS
LIN {X 0.112,Y -500.560,Z 391.474,A 0.000,B 0.000,C 90.000,E1 121.386} C_DIS
LIN {X -0.122,Y -497.438,Z 391.469,A 0.000,B 0.000,C 90.000,E1 120.512} C_DIS
LIN {X 0.036,Y -494.075,Z 391.464,A 0.000,B 0.000,C 90.000,E1 119.589} C_DIS
LIN {X -0.103,Y -491.664,Z 391.461,A 0.000,B 0.000,C 90.000,E1 118.999} C_DIS
LIN {X -0.248,Y -487.751,Z 391.456,A 0.000,B 0.000,C 90.000,E1 118.103} C_DIS
LIN {X 0.222,Y -483.672,Z 391.451,A 0.000,B 0.000,C 90.000,E1 117.129} C_DIS
LIN {X 0.167,Y -476.354,Z 391.442,A 0.000,B 0.000,C 90.000,E1 115.591} C_DIS
LIN {X 0.048,Y -471.069,Z 391.436,A 0.000,B 0.000,C 90.000,E1 114.515} C_DIS
LIN {X 0.161,Y -462.488,Z 391.427,A 0.000,B 0.000,C 90.000,E1 112.770} C_DIS
LIN {X 0.080,Y -453.851,Z 391.417,A 0.000,B 0.000,C 90.000,E1 111.046} C_DIS
LIN {X 0.040,Y -453.841,Z 391.417,A 0.000,B 0.000,C 90.000,E1 111.046} C_DIS
LIN {X -0.222,Y -456.976,Z 391.411,A 0.000,B 0.000,C 90.000,E1 109.939} C_DIS
LIN {X 0.015,Y -458.240,Z 391.407,A 0.000,B 0.000,C 90.000,E1 109.268} C_DIS
LIN {X 0.213,Y -466.398,Z 391.386,A 0.000,B 0.000,C 90.000,E1 105.426} C_DIS
LIN {X -0.062,Y -467.913,Z 391.382,A 0.000,B 0.000,C 90.000,E1 104.828} C_DIS
LIN {X -0.035,Y -475.484,Z 391.358,A 0.000,B 0.000,C 90.000,E1 100.433} C_DIS
LIN {X -0.197,Y -476.127,Z 391.356,A 0.000,B 0.000,C 90.000,E1 100.141} C_DIS
LIN {X 0.087,Y -482.042,Z 391.330,A 0.000,B 0.000,C 90.000,E1 95.454} C_DIS
LIN {X -0.123,Y -485.476,Z 391.305,A 0.000,B 0.000,C 90.000,E1 90.859} C_DIS
LIN {X 0.233,Y -486.108,Z 391.284,A 0.000,B 0.000,C 90.000,E1 87.135} C_DIS
LIN {X -0.091,Y -486.385,Z 391.281,A 0.000,B 0.000,C 90.000,E1 86.560} C_DIS
LIN {X 0.219,Y -486.364,Z 391.279,A 0.000,B 0.000,C 90.000,E1 86.216} C_DIS
LIN {X -0.178,Y -484.690,Z 391.254,A 0.000,B 0.000,C 90.000,E1 81.659} C_DIS
LIN {X -0.163,Y -483.694,Z 391.248,A 0.000,B 0.000,C 90.000,E1 80.735} C_DIS
LIN {X 0.202,Y -480.625,Z 391.228,A 0.000,B 0.000,C 90.000,E1 76.992} C_DIS
LIN {X 0.059,Y -480.302,Z 391.226,A 0.000,B 0.000,C 90.000,E1 76.700} C_DIS
LIN {X -0.036,Y -474.122,Z 391.200,A 0.000,B 0.000,C 90.000,E1 72.054} C_DIS
LIN {X 0.162,Y -472.266,Z 391.195,A 0.000,B 0.000,C 90.000,E1 71.094} C_DIS
LIN {X 0.122,Y -472.300,Z 391.195,A 0.000,B 0.000,C 90.000,E1 71.094} C_DIS
LIN {X 0.113,Y -482.439,Z 391.187,A 0.000,B 0.000,C 90.000,E1 69.699} C_DIS
LIN {X 0.159,Y -491.494,Z 391.181,A 0.000,B 0.000,C 90.000,E1 68.465} C_DIS
LIN {X 0.286,Y -497.947,Z 391.175,A 0.000,B 0.000,C 90.000,E1 67.539} C_DIS
LIN {X 0.217,Y -503.071,Z 391.171,A 0.000,B 0.000,C 90.000,E1 66.794} C_DIS
LIN {X -0.084,Y -507.155,Z 391.168,A 0.000,B 0.000,C 90.000,E1 66.230} C_DIS
LIN {X -0.074,Y -511.709,Z 391.164,A 0.000,B 0.000,C 90.000,E1 65.485} C_DIS
LIN {X 0.192,Y -515.936,Z 391.160,A 0.000,B 0.000,C 90.000,E1 64.717} C_DIS
LIN {X -0.189,Y -519.742,Z 391.156,A 0.000,B 0.000,C 90.000,E1 64.024} C_DIS
LIN {X -0.082,Y -522.511,Z 391.152,A 0.000,B 0.000,C 90.000,E1 63.435} C_DIS
LIN {X -0.116,Y -527.714,Z 391.146,A 0.000,B 0.000,C 90.000,E1 62.281} C_DIS
LIN {X -0.161,Y -530.476,Z 391.142,A 0.000,B 0.000,C 90.000,E1 61.563} C_DIS
LIN {X -0.037,Y -532.537,Z 391.139,A 0.000,B 0.000,C 90.000,E1 60.973} C_DIS
LIN {X -0.185,Y -535.188,Z 391.134,A 0.000,B 0.000,C 90.000,E1 60.127} C_DIS
LIN {X -0.026,Y -536.836,Z 391.131,A 0.000,B 0.000,C 90.000,E1 59.537} C_DIS
LIN {X -0.136,Y -540.441,Z 391.123,A 0.000,B 0.000,C 90.000,E1 58.122} C_DIS
LIN {X 0.055,Y -541.722,Z 391.120,A 0.000,B 0.000,C 90.000,E1 57.533} C_DIS
LIN {X -0.185,Y -543.240,Z 391.115,A 0.000,B 0.000,C 90.000,E1 56.707} C_DIS
LIN {X -0.132,Y -544.128,Z 391.112,A 0.000,B 0.000,C 90.000,E1 56.135} C_DIS
LIN {X 0.107,Y -545.146,Z 391.107,A 0.000,B 0.000,C 90.000,E1 55.261} C_DIS
LIN {X 0.218,Y -545.927,Z 391.102,A 0.000,B 0.000,C 90.000,E1 54.402} C_DIS
LIN {X -0.023,Y -546.174,Z 391.099,A 0.000,B 0.000,C 90.000,E1 53.863} C_DIS
LIN {X 0.141,Y -546.282,Z 391.093,A 0.000,B 0.000,C 90.000,E1 52.718} C_DIS
LIN {X -0.167,Y -546.082,Z 391.088,A 0.000,B 0.000,C 90.000,E1 51.904} C_DIS
LIN {X -0.086,Y -545.819,Z 391.085,A 0.000,B 0.000,C 90.000,E1 51.331} C_DIS
LIN {X 0.335,Y -545.439,Z 391.082,A 0.000,B 0.000,C 90.000,E1 50.723} C_DIS
LIN {X 0.056,Y -544.261,Z 391.076,A 0.000,B 0.000,C 90.000,E1 49.622} C_DIS
LIN {X 0.084,Y -543.200,Z 391.071,A 0.000,B 0.000,C 90.000,E1 48.771} C_DIS
LIN {X -0.263,Y -541.181,Z 391.063,A 0.000,B 0.000,C 90.000,E1 47.391} C_DIS
LIN {X 0.090,Y -538.557,Z 391.054,A 0.000,B 0.000,C 90.000,E1 45.648} C_DIS
LIN {X -0.012,Y -535.675,Z 391.043,A 0.000,B 0.000,C 90.000,E1 43.662} C_DIS
LIN {X 0.224,Y -533.402,Z 391.033,A 0.000,B 0.000,C 90.000,E1 41.919} C_DIS
LIN {X 0.020,Y -530.850,Z 391.022,A 0.000,B 0.000,C 90.000,E1 39.930} C_DIS
LIN {X 0.267,Y -529.001,Z 391.014,A 0.000,B 0.000,C 90.000,E1 38.463} C_DIS
LIN {X 0.160,Y -527.177,Z 391.006,A 0.000,B 0.000,C 90.000,E1 37.030} C_DIS
LIN {X -0.011,Y -524.887,Z 390.996,A 0.000,B 0.000,C 90.000,E1 35.311} C_DIS
LIN {X -0.156,Y -522.215,Z 390.985,A 0.000,B 0.000,C 90.000,E1 33.293} C_DIS
LIN {X -0.224,Y -519.506,Z 390.974,A 0.000,B 0.000,C 90.000,E1 31.258} C_DIS
LIN {X -0.186,Y -516.891,Z 390.962,A 0.000,B 0.000,C 90.000,E1 29.205} C_DIS
LIN {X -0.012,Y -514.385,Z 390.951,A 0.000,B 0.000,C 90.000,E1 27.129} C_DIS
LIN {X 0.210,Y -512.436,Z 390.941,A 0.000,B 0.000,C 90.000,E1 25.335} C_DIS
LIN {X -0.087,Y -510.041,Z 390.928,A 0.000,B 0.000,C 90.000,E1 23.003} C_DIS
LIN {X -0.111,Y -508.428,Z 390.918,A 0.000,B 0.000,C 90.000,E1 21.227} C_DIS
LIN {X -0.068,Y -506.879,Z 390.906,A 0.000,B 0.000,C 90.000,E1 19.141} C_DIS
LIN {X 0.081,Y -505.474,Z 390.895,A 0.000,B 0.000,C 90.000,E1 17.040} C_DIS
LIN {X 0.118,Y -504.475,Z 390.885,A 0.000,B 0.000,C 90.000,E1 15.245} C_DIS
LIN {X -0.070,Y -503.580,Z 390.873,A 0.000,B 0.000,C 90.000,E1 13.175} C_DIS
LIN {X -0.261,Y -502.794,Z 390.855,A 0.000,B 0.000,C 90.000,E1 9.905} C_DIS
LIN {X -0.235,Y -502.764,Z 390.845,A 0.000,B 0.000,C 90.000,E1 8.106} C_DIS
LIN {X 0.017,Y -503.205,Z 390.832,A 0.000,B 0.000,C 90.000,E1 5.682} C_DIS
LIN {X 0.193,Y -505.174,Z 390.810,A 0.000,B 0.000,C 90.000,E1 1.776} C_DIS
LIN {X 0.206,Y -508.482,Z 390.791,A 0.000,B 0.000,C 90.000,E1 358.282} C_DIS
LIN {X -0.223,Y -510.376,Z 390.782,A 0.000,B 0.000,C 90.000,E1 356.846} C_DIS
LIN {X 0.047,Y -511.529,Z 390.777,A 0.000,B 0.000,C 90.000,E1 355.927} C_DIS
LIN {X 0.199,Y -513.821,Z 390.769,A 0.000,B 0.000,C 90.000,E1 354.432} C_DIS
LIN {X -0.156,Y -516.804,Z 390.759,A 0.000,B 0.000,C 90.000,E1 352.704} C_DIS
LIN {X 0.114,Y -521.222,Z 390.746,A 0.000,B 0.000,C 90.000,E1 350.330} C_DIS
LIN {X -0.208,Y -529.957,Z 390.725,A 0.000,B 0.000,C 90.000,E1 346.589} C_DIS
LIN {X -0.201,Y -535.284,Z 390.714,A 0.000,B 0.000,C 90.000,E1 344.574} C_DIS
LIN {X 0.036,Y -539.982,Z 390.705,A 0.000,B 0.000,C 90.000,E1 342.834} C_DIS
LIN {X -0.135,Y -544.712,Z 390.695,A 0.000,B 0.000,C 90.000,E1 341.148} C_DIS
LIN {X 0.227,Y -548.775,Z 390.687,A 0.000,B 0.000,C 90.000,E1 339.699} C_DIS
LIN {X 0.100,Y -553.647,Z 390.678,A 0.000,B 0.000,C 90.000,E1 338.028} C_DIS
LIN {X -0.216,Y -557.830,Z 390.670,A 0.000,B 0.000,C 90.000,E1 336.666} C_DIS
LIN {X 0.072,Y -562.849,Z 390.661,A 0.000,B 0.000,C 90.000,E1 334.973} C_DIS
LIN {X -0.154,Y -569.696,Z 390.649,A 0.000,B 0.000,C 90.000,E1 332.794} C_DIS
LIN {X -0.079,Y -577.734,Z 390.635,A 0.000,B 0.000,C 90.000,E1 330.333} C_DIS
LIN {X -0.236,Y -582.198,Z 390.628,A 0.000,B 0.000,C 90.000,E1 328.997} C_DIS
LIN {X -0.317,Y -586.715,Z 390.620,A 0.000,B 0.000,C 90.000,E1 327.661} C_DIS
LIN {X -0.209,Y -593.946,Z 390.608,A 0.000,B 0.000,C 90.000,E1 325.515} C_DIS
LIN {X -0.029,Y -599.437,Z 390.600,A 0.000,B 0.000,C 90.000,E1 323.909} C_DIS
LIN {X 0.030,Y -606.061,Z 390.589,A 0.000,B 0.000,C 90.000,E1 322.065} C_DIS
LIN {X 0.130,Y -612.707,Z 390.579,A 0.000,B 0.000,C 90.000,E1 320.231} C_DIS
LIN {X 0.182,Y -617.518,Z 390.572,A 0.000,B 0.000,C 90.000,E1 318.933} C_DIS
LIN {X -0.141,Y -622.183,Z 390.565,A 0.000,B 0.000,C 90.000,E1 317.676} C_DIS
LIN {X 0.208,Y -625.903,Z 390.559,A 0.000,B 0.000,C 90.000,E1 316.620} C_DIS
LIN {X 0.229,Y -632.266,Z 390.549,A 0.000,B 0.000,C 90.000,E1 314.838} C_DIS
LIN {X -0.306,Y -636.874,Z 390.542,A 0.000,B 0.000,C 90.000,E1 313.623} C_DIS
LIN {X 0.079,Y -642.457,Z 390.534,A 0.000,B 0.000,C 90.000,E1 312.081} C_DIS
LIN {X -0.331,Y -647.958,Z 390.526,A 0.000,B 0.000,C 90.000,E1 310.620} C_DIS
LIN {X 0.390,Y -651.472,Z 390.520,A 0.000,B 0.000,C 90.000,E1 309.564} C_DIS
LIN {X -0.171,Y -654.916,Z 390.515,A 0.000,B 0.000,C 90.000,E1 308.624} C_DIS
LIN {X 0.238,Y -658.252,Z 390.509,A 0.000,B 0.000,C 90.000,E1 307.604} C_DIS
LIN {X -0.192,Y -662.984,Z 390.501,A 0.000,B 0.000,C 90.000,E1 306.171} C_DIS
LIN {X -0.118,Y -666.768,Z 390.494,A 0.000,B 0.000,C 90.000,E1 304.945} C_DIS
LIN {X -0.333,Y -669.664,Z 390.489,A 0.000,B 0.000,C 90.000,E1 303.992} C_DIS
LIN {X 0.174,Y -673.966,Z 390.481,A 0.000,B 0.000,C 90.000,E1 302.498} C_DIS
LIN {X 0.061,Y -676.752,Z 390.475,A 0.000,B 0.000,C 90.000,E1 301.544} C_DIS
LIN {X -0.230,Y -680.640,Z 390.467,A 0.000,B 0.000,C 90.000,E1 300.129} C_DIS
LIN {X -0.227,Y -682.463,Z 390.463,A 0.000,B 0.000,C 90.000,E1 299.411} C_DIS
LIN {X 0.008,Y -684.447,Z 390.458,A 0.000,B 0.000,C 90.000,E1 298.437} C_DIS
LIN {X -0.336,Y -686.075,Z 390.453,A 0.000,B 0.000,C 90.000,E1 297.513} C_DIS
LIN {X 0.164,Y -687.584,Z 390.446,A 0.000,B 0.000,C 90.000,E1 296.283} C_DIS
LIN {X -0.076,Y -688.430,Z 390.442,A 0.000,B 0.000,C 90.000,E1 295.591} C_DIS
LIN {X -0.305,Y -688.911,Z 390.438,A 0.000,B 0.000,C 90.000,E1 294.899} C_DIS
LIN {X -0.070,Y -689.237,Z 390.432,A 0.000,B 0.000,C 90.000,E1 293.695} C_DIS
LIN {X -0.337,Y -688.961,Z 390.426,A 0.000,B 0.000,C 90.000,E1 292.770} C_DIS
LIN {X 0.073,Y -688.628,Z 390.422,A 0.000,B 0.000,C 90.000,E1 292.025} C_DIS
LIN {X -0.163,Y -688.063,Z 390.418,A 0.000,B 0.000,C 90.000,E1 291.334} C_DIS
LIN {X -0.046,Y -686.853,Z 390.413,A 0.000,B 0.000,C 90.000,E1 290.375} C_DIS
LIN {X 0.334,Y -685.777,Z 390.409,A 0.000,B 0.000,C 90.000,E1 289.631} C_DIS
LIN {X -0.240,Y -683.851,Z 390.403,A 0.000,B 0.000,C 90.000,E1 288.489} C_DIS
LIN {X 0.056,Y -682.210,Z 390.397,A 0.000,B 0.000,C 90.000,E1 287.511} C_DIS
LIN {X -0.045,Y -680.939,Z 390.393,A 0.000,B 0.000,C 90.000,E1 286.804} C_DIS
LIN {X -0.037,Y -678.826,Z 390.387,A 0.000,B 0.000,C 90.000,E1 285.607} C_DIS
LIN {X -0.028,Y -677.023,Z 390.381,A 0.000,B 0.000,C 90.000,E1 284.647} C_DIS
LIN {X 0.276,Y -673.992,Z 390.372,A 0.000,B 0.000,C 90.000,E1 282.939} C_DIS
LIN {X 0.105,Y -670.410,Z 390.360,A 0.000,B 0.000,C 90.000,E1 280.782} C_DIS
LIN {X -0.161,Y -667.452,Z 390.348,A 0.000,B 0.000,C 90.000,E1 278.624} C_DIS
LIN {X 0.128,Y -664.500,Z 390.332,A 0.000,B 0.000,C 90.000,E1 275.682} C_DIS
LIN {X -0.155,Y -662.992,Z 390.318,A 0.000,B 0.000,C 90.000,E1 273.269} C_DIS
LIN {X 0.142,Y -662.357,Z 390.305,A 0.000,B 0.000,C 90.000,E1 270.802} C_DIS
LIN {X -0.240,Y -661.939,Z 390.296,A 0.000,B 0.000,C 90.000,E1 269.370} C_DIS
LIN {X -0.283,Y -661.753,Z 390.291,A 0.000,B 0.000,C 90.000,E1 268.396} C_DIS
LIN {X 0.142,Y -661.194,Z 390.279,A 0.000,B 0.000,C 90.000,E1 266.159} C_DIS
LIN {X 0.163,Y -660.844,Z 390.273,A 0.000,B 0.000,C 90.000,E1 265.179} C_DIS
LIN {X 0.125,Y -660.017,Z 390.268,A 0.000,B 0.000,C 90.000,E1 264.204} C_DIS
LIN {X 0.261,Y -659.161,Z 390.264,A 0.000,B 0.000,C 90.000,E1 263.457} C_DIS
LIN {X 0.131,Y -657.330,Z 390.257,A 0.000,B 0.000,C 90.000,E1 262.243} C_DIS
LIN {X -0.025,Y -654.997,Z 390.250,A 0.000,B 0.000,C 90.000,E1 261.027} C_DIS
LIN {X 0.013,Y -652.878,Z 390.245,A 0.000,B 0.000,C 90.000,E1 260.038} C_DIS
LIN {X -0.112,Y -652.247,Z 390.243,A 0.000,B 0.000,C 90.000,E1 259.803} C_DIS
LIN {X 0.154,Y -651.232,Z 390.241,A 0.000,B 0.000,C 90.000,E1 259.285} C_DIS
LIN {X 0.266,Y -648.846,Z 390.235,A 0.000,B 0.000,C 90.000,E1 258.285} C_DIS
LIN {X 0.074,Y -645.668,Z 390.228,A 0.000,B 0.000,C 90.000,E1 257.061} C_DIS
LIN {X -0.360,Y -643.565,Z 390.224,A 0.000,B 0.000,C 90.000,E1 256.353} C_DIS
LIN {X -0.029,Y -641.434,Z 390.220,A 0.000,B 0.000,C 90.000,E1 255.574} C_DIS
LIN {X -0.206,Y -637.560,Z 390.213,A 0.000,B 0.000,C 90.000,E1 254.338} C_DIS
LIN {X -0.105,Y -634.139,Z 390.207,A 0.000,B 0.000,C 90.000,E1 253.323} C_DIS
LIN {X -0.052,Y -630.562,Z 390.202,A 0.000,B 0.000,C 90.000,E1 252.308} C_DIS
LIN {X 0.144,Y -626.843,Z 390.196,A 0.000,B 0.000,C 90.000,E1 251.275} C_DIS
LIN {X 0.294,Y -622.890,Z 390.190,A 0.000,B 0.000,C 90.000,E1 250.242} C_DIS
LIN {X 0.144,Y -617.843,Z 390.183,A 0.000,B 0.000,C 90.000,E1 248.975} C_DIS
LIN {X -0.217,Y -612.609,Z 390.176,A 0.000,B 0.000,C 90.000,E1 247.720} C_DIS
LIN {X -0.039,Y -608.316,Z 390.170,A 0.000,B 0.000,C 90.000,E1 246.666} C_DIS
LIN {X -0.048,Y -601.667,Z 390.162,A 0.000,B 0.000,C 90.000,E1 245.101} C_DIS
LIN {X 0.217,Y -597.233,Z 390.156,A 0.000,B 0.000,C 90.000,E1 244.024} C_DIS
LIN {X -0.305,Y -590.570,Z 390.147,A 0.000,B 0.000,C 90.000,E1 242.487} C_DIS
LIN {X 0.112,Y -583.934,Z 390.138,A 0.000,B 0.000,C 90.000,E1 240.845} C_DIS
LIN {X -0.257,Y -576.462,Z 390.128,A 0.000,B 0.000,C 90.000,E1 238.997} C_DIS
LIN {X 0.327,Y -566.450,Z 390.113,A 0.000,B 0.000,C 90.000,E1 236.215} C_DIS
LIN {X -0.019,Y -559.846,Z 390.102,A 0.000,B 0.000,C 90.000,E1 234.322} C_DIS
LIN {X 0.015,Y -556.183,Z 390.096,A 0.000,B 0.000,C 90.000,E1 233.210} C_DIS
LIN {X -0.050,Y -551.447,Z 390.088,A 0.000,B 0.000,C 90.000,E1 231.823} C_DIS
LIN {X -0.151,Y -545.713,Z 390.079,A 0.000,B 0.000,C 90.000,E1 230.150} C_DIS
LIN {X -0.060,Y -540.992,Z 390.071,A 0.000,B 0.000,C 90.000,E1 228.728} C_DIS
LIN {X -0.097,Y -536.442,Z 390.063,A 0.000,B 0.000,C 90.000,E1 227.310} C_DIS
LIN {X 0.135,Y -531.124,Z 390.053,A 0.000,B 0.000,C 90.000,E1 225.567} C_DIS
LIN {X 0.187,Y -524.901,Z 390.042,A 0.000,B 0.000,C 90.000,E1 223.542} C_DIS
LIN {X 0.094,Y -518.906,Z 390.031,A 0.000,B 0.000,C 90.000,E1 221.515} C_DIS
LIN {X -0.182,Y -512.249,Z 390.018,A 0.000,B 0.000,C 90.000,E1 219.197} C_DIS
LIN {X 0.119,Y -508.254,Z 390.009,A 0.000,B 0.000,C 90.000,E1 217.684} C_DIS
LIN {X 0.024,Y -502.101,Z 389.996,A 0.000,B 0.000,C 90.000,E1 215.311} C_DIS
LIN {X 0.118,Y -497.601,Z 389.986,A 0.000,B 0.000,C 90.000,E1 213.499} C_DIS
LIN {X -0.017,Y -494.057,Z 389.978,A 0.000,B 0.000,C 90.000,E1 212.005} C_DIS
LIN {X -0.216,Y -489.828,Z 389.968,A 0.000,B 0.000,C 90.000,E1 210.207} C_DIS
LIN {X -0.085,Y -485.606,Z 389.958,A 0.000,B 0.000,C 90.000,E1 208.359} C_DIS
LIN {X -0.067,Y -482.776,Z 389.951,A 0.000,B 0.000,C 90.000,E1 207.129} C_DIS
LIN {X -0.108,Y -479.095,Z 389.942,A 0.000,B 0.000,C 90.000,E1 205.591} C_DIS
LIN {X 0.011,Y -475.437,Z 389.934,A 0.000,B 0.000,C 90.000,E1 204.027} C_DIS
LIN {X 0.062,Y -471.612,Z 389.925,A 0.000,B 0.000,C 90.000,E1 202.461} C_DIS
LIN {X -0.141,Y -467.898,Z 389.916,A 0.000,B 0.000,C 90.000,E1 200.918} C_DIS
LIN {X 0.167,Y -462.805,Z 389.904,A 0.000,B 0.000,C 90.000,E1 198.671} C_DIS
LIN {X 0.190,Y -458.135,Z 389.892,A 0.000,B 0.000,C 90.000,E1 196.441} C_DIS
LIN {X -0.091,Y -452.552,Z 389.875,A 0.000,B 0.000,C 90.000,E1 193.592} C_DIS
LIN {X -0.086,Y -447.943,Z 389.861,A 0.000,B 0.000,C 90.000,E1 191.007} C_DIS
LIN {X -0.206,Y -444.240,Z 389.848,A 0.000,B 0.000,C 90.000,E1 188.746} C_DIS
LIN {X 0.015,Y -440.844,Z 389.836,A 0.000,B 0.000,C 90.000,E1 186.429} C_DIS
LIN {X 0.021,Y -436.366,Z 389.816,A 0.000,B 0.000,C 90.000,E1 182.808} C_DIS
LIN {X -0.052,Y -432.704,Z 389.792,A 0.000,B 0.000,C 90.000,E1 178.511} C_DIS
LIN {X -0.202,Y -430.952,Z 389.768,A 0.000,B 0.000,C 90.000,E1 174.204} C_DIS
LIN {X 0.104,Y -431.087,Z 389.740,A 0.000,B 0.000,C 90.000,E1 169.162} C_DIS
LIN {X -0.018,Y -433.632,Z 389.714,A 0.000,B 0.000,C 90.000,E1 164.519} C_DIS
LIN {X 0.107,Y -435.765,Z 389.701,A 0.000,B 0.000,C 90.000,E1 162.181} C_DIS
LIN {X -0.053,Y -439.676,Z 389.683,A 0.000,B 0.000,C 90.000,E1 158.901} C_DIS
LIN {X -0.091,Y -445.627,Z 389.661,A 0.000,B 0.000,C 90.000,E1 154.973} C_DIS
LIN {X -0.042,Y -451.649,Z 389.643,A 0.000,B 0.000,C 90.000,E1 151.719} C_DIS
LIN {X -0.021,Y -458.155,Z 389.627,A 0.000,B 0.000,C 90.000,E1 148.820} C_DIS
LIN {X -0.208,Y -464.801,Z 389.613,A 0.000,B 0.000,C 90.000,E1 146.294} C_DIS
LIN {X 0.130,Y -473.250,Z 389.597,A 0.000,B 0.000,C 90.000,E1 143.417} C_DIS
LIN {X -0.191,Y -481.419,Z 389.583,A 0.000,B 0.000,C 90.000,E1 140.964} C_DIS
LIN {X 0.173,Y -486.578,Z 389.574,A 0.000,B 0.000,C 90.000,E1 139.380} C_DIS
LIN {X -0.052,Y -491.676,Z 389.566,A 0.000,B 0.000,C 90.000,E1 137.877} C_DIS
LIN {X -0.065,Y -495.517,Z 389.559,A 0.000,B 0.000,C 90.000,E1 136.662} C_DIS
LIN {X -0.001,Y -499.080,Z 389.553,A 0.000,B 0.000,C 90.000,E1 135.445} C_DIS
LIN {X -0.251,Y -502.448,Z 389.546,A 0.000,B 0.000,C 90.000,E1 134.271} C_DIS
LIN {X -0.100,Y -505.305,Z 389.539,A 0.000,B 0.000,C 90.000,E1 133.056} C_DIS
LIN {X 0.120,Y -507.882,Z 389.533,A 0.000,B 0.000,C 90.000,E1 131.838} C_DIS
LIN {X -0.237,Y -509.470,Z 389.528,A 0.000,B 0.000,C 90.000,E1 130.987} C_DIS
LIN {X -0.193,Y -510.855,Z 389.523,A 0.000,B 0.000,C 90.000,E1 130.092} C_DIS
LIN {X -0.132,Y -511.844,Z 389.518,A 0.000,B 0.000,C 90.000,E1 129.197} C_DIS
LIN {X -0.062,Y -512.538,Z 389.513,A 0.000,B 0.000,C 90.000,E1 128.302} C_DIS
LIN {X -0.302,Y -512.574,Z 389.508,A 0.000,B 0.000,C 90.000,E1 127.443} C_DIS
LIN {X 0.177,Y -512.066,Z 389.503,A 0.000,B 0.000,C 90.000,E1 126.503} C_DIS
LIN {X -0.069,Y -511.183,Z 389.498,A 0.000,B 0.000,C 90.000,E1 125.644} C_DIS
LIN {X 0.090,Y -509.982,Z 389.493,A 0.000,B 0.000,C 90.000,E1 124.739} C_DIS
LIN {X 0.330,Y -509.029,Z 389.490,A 0.000,B 0.000,C 90.000,E1 124.119} C_DIS
LIN {X -0.239,Y -507.120,Z 389.485,A 0.000,B 0.000,C 90.000,E1 123.293} C_DIS
LIN {X -0.021,Y -505.705,Z 389.482,A 0.000,B 0.000,C 90.000,E1 122.673} C_DIS
LIN {X 0.110,Y -502.264,Z 389.475,A 0.000,B 0.000,C 90.000,E1 121.465} C_DIS
LIN {X 0.029,Y -500.311,Z 389.472,A 0.000,B 0.000,C 90.000,E1 120.875} C_DIS
LIN {X -0.204,Y -497.114,Z 389.467,A 0.000,B 0.000,C 90.000,E1 120.001} C_DIS
LIN {X -0.044,Y -493.640,Z 389.462,A 0.000,B 0.000,C 90.000,E1 119.077} C_DIS
LIN {X 0.067,Y -489.790,Z 389.457,A 0.000,B 0.000,C 90.000,E1 118.153} C_DIS
LIN {X 0.121,Y -485.082,Z 389.451,A 0.000,B 0.000,C 90.000,E1 117.078} C_DIS
LIN {X 0.099,Y -477.782,Z 389.442,A 0.000,B 0.000,C 90.000,E1 115.540} C_DIS
LIN {X 0.006,Y -472.547,Z 389.436,A 0.000,B 0.000,C 90.000,E1 114.463} C_DIS
LIN {X 0.078,Y -467.794,Z 389.431,A 0.000,B 0.000,C 90.000,E1 113.515} C_DIS
LIN {X -0.090,Y -463.130,Z 389.425,A 0.000,B 0.000,C 90.000,E1 112.589} C_DIS
LIN {X 0.115,Y -455.183,Z 389.417,A 0.000,B 0.000,C 90.000,E1 110.972} C_DIS
LIN {X -0.067,Y -454.436,Z 389.416,A 0.000,B 0.000,C 90.000,E1 110.844} C_DIS
LIN {X -0.107,Y -454.429,Z 389.416,A 0.000,B 0.000,C 90.000,E1 110.844} C_DIS
LIN {X 0.239,Y -456.659,Z 389.411,A 0.000,B 0.000,C 90.000,E1 109.993} C_DIS
LIN {X -0.015,Y -457.465,Z 389.410,A 0.000,B 0.000,C 90.000,E1 109.704} C_DIS
LIN {X 0.086,Y -466.129,Z 389.387,A 0.000,B 0.000,C 90.000,E1 105.552} C_DIS
LIN {X -0.190,Y -467.699,Z 389.383,A 0.000,B 0.000,C 90.000,E1 104.954} C_DIS
LIN {X -0.233,Y -475.909,Z 389.357,A 0.000,B 0.000,C 90.000,E1 100.254} C_DIS
LIN {X 0.075,Y -476.353,Z 389.355,A 0.000,B 0.000,C 90.000,E1 99.905} C_DIS
LIN {X 0.030,Y -481.871,Z 389.331,A 0.000,B 0.000,C 90.000,E1 95.568} C_DIS
LIN {X -0.122,Y -482.192,Z 389.329,A 0.000,B 0.000,C 90.000,E1 95.277} C_DIS
LIN {X -0.188,Y -485.362,Z 389.305,A 0.000,B 0.000,C 90.000,E1 90.974} C_DIS
LIN {X 0.121,Y -485.532,Z 389.304,A 0.000,B 0.000,C 90.000,E1 90.630} C_DIS
LIN {X -0.156,Y -486.344,Z 389.281,A 0.000,B 0.000,C 90.000,E1 86.674} C_DIS
LIN {X -0.022,Y -486.270,Z 389.278,A 0.000,B 0.000,C 90.000,E1 86.045} C_DIS
LIN {X 0.177,Y -484.693,Z 389.254,A 0.000,B 0.000,C 90.000,E1 81.724} C_DIS
LIN {X 0.046,Y -484.538,Z 389.252,A 0.000,B 0.000,C 90.000,E1 81.432} C_DIS
LIN {X -0.084,Y -480.476,Z 389.227,A 0.000,B 0.000,C 90.000,E1 76.825} C_DIS
LIN {X -0.187,Y -474.234,Z 389.201,A 0.000,B 0.000,C 90.000,E1 72.181} C_DIS
LIN {X 0.231,Y -473.741,Z 389.199,A 0.000,B 0.000,C 90.000,E1 71.819} C_DIS
LIN {X -0.159,Y -472.652,Z 389.196,A 0.000,B 0.000,C 90.000,E1 71.329} C_DIS
LIN {X 0.249,Y -472.644,Z 389.196,A 0.000,B 0.000,C 90.000,E1 71.275} C_DIS
LIN {X -0.254,Y -482.226,Z 389.189,A 0.000,B 0.000,C 90.000,E1 70.007} C_DIS
LIN {X -0.222,Y -491.242,Z 389.182,A 0.000,B 0.000,C 90.000,E1 68.773} C_DIS
LIN {X -0.151,Y -495.585,Z 389.179,A 0.000,B 0.000,C 90.000,E1 68.156} C_DIS
LIN {X -0.176,Y -502.812,Z 389.173,A 0.000,B 0.000,C 90.000,E1 67.102} C_DIS
LIN {X -0.206,Y -507.715,Z 389.169,A 0.000,B 0.000,C 90.000,E1 66.357} C_DIS
LIN {X -0.012,Y -511.317,Z 389.165,A 0.000,B 0.000,C 90.000,E1 65.741} C_DIS
LIN {X -0.043,Y -514.576,Z 389.162,A 0.000,B 0.000,C 90.000,E1 65.153} C_DIS
LIN {X -0.094,Y -517.004,Z 389.160,A 0.000,B 0.000,C 90.000,E1 64.717} C_DIS
LIN {X 0.165,Y -519.951,Z 389.156,A 0.000,B 0.000,C 90.000,E1 64.101} C_DIS
LIN {X 0.113,Y -523.234,Z 389.152,A 0.000,B 0.000,C 90.000,E1 63.384} C_DIS
LIN {X 0.099,Y -525.080,Z 389.150,A 0.000,B 0.000,C 90.000,E1 62.948} C_DIS
LIN {X 0.179,Y -527.465,Z 389.147,A 0.000,B 0.000,C 90.000,E1 62.359} C_DIS
LIN {X 0.024,Y -528.113,Z 389.146,A 0.000,B 0.000,C 90.000,E1 62.231} C_DIS
LIN {X 0.130,Y -530.240,Z 389.143,A 0.000,B 0.000,C 90.000,E1 61.641} C_DIS
LIN {X -0.044,Y -533.187,Z 389.138,A 0.000,B 0.000,C 90.000,E1 60.795} C_DIS
LIN {X 0.078,Y -535.757,Z 389.133,A 0.000,B 0.000,C 90.000,E1 59.921} C_DIS
LIN {X 0.242,Y -537.342,Z 389.130,A 0.000,B 0.000,C 90.000,E1 59.331} C_DIS
LIN {X 0.138,Y -540.261,Z 389.123,A 0.000,B 0.000,C 90.000,E1 58.201} C_DIS
LIN {X -0.115,Y -542.107,Z 389.119,A 0.000,B 0.000,C 90.000,E1 57.375} C_DIS
LIN {X 0.107,Y -543.664,Z 389.114,A 0.000,B 0.000,C 90.000,E1 56.501} C_DIS
LIN {X -0.140,Y -544.570,Z 389.111,A 0.000,B 0.000,C 90.000,E1 55.960} C_DIS
LIN {X -0.039,Y -545.632,Z 389.106,A 0.000,B 0.000,C 90.000,E1 55.102} C_DIS
LIN {X -0.239,Y -546.438,Z 389.101,A 0.000,B 0.000,C 90.000,E1 54.276} C_DIS
LIN {X -0.155,Y -546.642,Z 389.098,A 0.000,B 0.000,C 90.000,E1 53.703} C_DIS
LIN {X -0.111,Y -546.610,Z 389.097,A 0.000,B 0.000,C 90.000,E1 53.417} C_DIS
LIN {X 0.020,Y -546.944,Z 389.092,A 0.000,B 0.000,C 90.000,E1 52.557} C_DIS
LIN {X -0.233,Y -546.697,Z 389.086,A 0.000,B 0.000,C 90.000,E1 51.457} C_DIS
LIN {X -0.108,Y -546.194,Z 389.081,A 0.000,B 0.000,C 90.000,E1 50.598} C_DIS
LIN {X -0.063,Y -545.377,Z 389.076,A 0.000,B 0.000,C 90.000,E1 49.747} C_DIS
LIN {X 0.012,Y -543.969,Z 389.070,A 0.000,B 0.000,C 90.000,E1 48.609} C_DIS
LIN {X 0.063,Y -542.343,Z 389.064,A 0.000,B 0.000,C 90.000,E1 47.472} C_DIS
LIN {X 0.064,Y -540.204,Z 389.056,A 0.000,B 0.000,C 90.000,E1 46.053} C_DIS
LIN {X -0.022,Y -536.858,Z 389.043,A 0.000,B 0.000,C 90.000,E1 43.785} C_DIS
LIN {X -0.129,Y -534.565,Z 389.034,A 0.000,B 0.000,C 90.000,E1 42.081} C_DIS
LIN {X 0.031,Y -531.648,Z 389.021,A 0.000,B 0.000,C 90.000,E1 39.769} C_DIS
LIN {X -0.039,Y -529.775,Z 389.013,A 0.000,B 0.000,C 90.000,E1 38.338} C_DIS
LIN {X 0.213,Y -528.313,Z 389.007,A 0.000,B 0.000,C 90.000,E1 37.156} C_DIS
LIN {X 0.061,Y -526.047,Z 388.997,A 0.000,B 0.000,C 90.000,E1 35.438} C_DIS
LIN {X -0.062,Y -523.362,Z 388.986,A 0.000,B 0.000,C 90.000,E1 33.420} C_DIS
LIN {X -0.104,Y -520.664,Z 388.974,A 0.000,B 0.000,C 90.000,E1 31.386} C_DIS
LIN {X 0.039,Y -518.427,Z 388.965,A 0.000,B 0.000,C 90.000,E1 29.617} C_DIS
LIN {X -0.195,Y -515.929,Z 388.953,A 0.000,B 0.000,C 90.000,E1 27.590} C_DIS
LIN {X -0.052,Y -513.618,Z 388.942,A 0.000,B 0.000,C 90.000,E1 25.515} C_DIS
LIN {X -0.167,Y -511.478,Z 388.930,A 0.000,B 0.000,C 90.000,E1 23.462} C_DIS
LIN {X 0.042,Y -509.867,Z 388.920,A 0.000,B 0.000,C 90.000,E1 21.663} C_DIS
LIN {X 0.229,Y -508.018,Z 388.907,A 0.000,B 0.000,C 90.000,E1 19.268} C_DIS
LIN {X -0.071,Y -506.612,Z 388.896,A 0.000,B 0.000,C 90.000,E1 17.221} C_DIS
LIN {X -0.064,Y -505.486,Z 388.884,A 0.000,B 0.000,C 90.000,E1 15.134} C_DIS
LIN {X -0.275,Y -504.510,Z 388.871,A 0.000,B 0.000,C 90.000,E1 12.771} C_DIS
LIN {X 0.024,Y -503.926,Z 388.851,A 0.000,B 0.000,C 90.000,E1 9.151} C_DIS
LIN {X 0.116,Y -504.365,Z 388.833,A 0.000,B 0.000,C 90.000,E1 5.853} C_DIS
LIN {X 0.237,Y -506.498,Z 388.809,A 0.000,B 0.000,C 90.000,E1 1.661} C_DIS
LIN {X 0.230,Y -509.765,Z 388.791,A 0.000,B 0.000,C 90.000,E1 358.282} C_DIS
LIN {X -0.176,Y -511.689,Z 388.782,A 0.000,B 0.000,C 90.000,E1 356.846} C_DIS
LIN {X 0.161,Y -512.373,Z 388.779,A 0.000,B 0.000,C 90.000,E1 356.216} C_DIS
LIN {X -0.063,Y -513.790,Z 388.774,A 0.000,B 0.000,C 90.000,E1 355.355} C_DIS
LIN {X -0.019,Y -517.627,Z 388.761,A 0.000,B 0.000,C 90.000,E1 352.996} C_DIS
LIN {X -0.243,Y -521.437,Z 388.750,A 0.000,B 0.000,C 90.000,E1 350.971} C_DIS
LIN {X -0.044,Y -529.918,Z 388.729,A 0.000,B 0.000,C 90.000,E1 347.173} C_DIS
LIN {X -0.168,Y -535.170,Z 388.718,A 0.000,B 0.000,C 90.000,E1 345.172} C_DIS
LIN {X 0.120,Y -540.674,Z 388.706,A 0.000,B 0.000,C 90.000,E1 343.142} C_DIS
LIN {X 0.202,Y -546.222,Z 388.695,A 0.000,B 0.000,C 90.000,E1 341.148} C_DIS
LIN {X 0.079,Y -550.306,Z 388.688,A 0.000,B 0.000,C 90.000,E1 339.752} C_DIS
LIN {X 0.067,Y -556.026,Z 388.677,A 0.000,B 0.000,C 90.000,E1 337.794} C_DIS
LIN {X 0.007,Y -560.194,Z 388.669,A 0.000,B 0.000,C 90.000,E1 336.410} C_DIS
LIN {X 0.351,Y -565.220,Z 388.660,A 0.000,B 0.000,C 90.000,E1 334.717} C_DIS
LIN {X 0.106,Y -571.221,Z 388.649,A 0.000,B 0.000,C 90.000,E1 332.820} C_DIS
LIN {X -0.139,Y -578.344,Z 388.637,A 0.000,B 0.000,C 90.000,E1 330.667} C_DIS
LIN {X 0.373,Y -583.746,Z 388.628,A 0.000,B 0.000,C 90.000,E1 328.997} C_DIS
LIN {X -0.174,Y -588.251,Z 388.621,A 0.000,B 0.000,C 90.000,E1 327.709} C_DIS
LIN {X 0.145,Y -595.478,Z 388.609,A 0.000,B 0.000,C 90.000,E1 325.548} C_DIS
LIN {X -0.139,Y -600.992,Z 388.600,A 0.000,B 0.000,C 90.000,E1 323.989} C_DIS
LIN {X -0.048,Y -607.610,Z 388.590,A 0.000,B 0.000,C 90.000,E1 322.145} C_DIS
LIN {X -0.385,Y -614.274,Z 388.580,A 0.000,B 0.000,C 90.000,E1 320.356} C_DIS
LIN {X 0.164,Y -619.083,Z 388.572,A 0.000,B 0.000,C 90.000,E1 319.013} C_DIS
LIN {X -0.134,Y -623.758,Z 388.565,A 0.000,B 0.000,C 90.000,E1 317.757} C_DIS
LIN {X 0.236,Y -627.494,Z 388.560,A 0.000,B 0.000,C 90.000,E1 316.701} C_DIS
LIN {X 0.295,Y -633.842,Z 388.550,A 0.000,B 0.000,C 90.000,E1 314.919} C_DIS
LIN {X -0.213,Y -638.454,Z 388.543,A 0.000,B 0.000,C 90.000,E1 313.704} C_DIS
LIN {X 0.204,Y -644.029,Z 388.534,A 0.000,B 0.000,C 90.000,E1 312.162} C_DIS
LIN {X -0.173,Y -649.538,Z 388.526,A 0.000,B 0.000,C 90.000,E1 310.701} C_DIS
LIN {X 0.100,Y -653.933,Z 388.519,A 0.000,B 0.000,C 90.000,E1 309.439} C_DIS
LIN {X 0.035,Y -656.521,Z 388.515,A 0.000,B 0.000,C 90.000,E1 308.705} C_DIS
LIN {X 0.423,Y -660.669,Z 388.508,A 0.000,B 0.000,C 90.000,E1 307.443} C_DIS
LIN {X 0.033,Y -665.362,Z 388.500,A 0.000,B 0.000,C 90.000,E1 306.011} C_DIS
LIN {X 0.181,Y -668.356,Z 388.495,A 0.000,B 0.000,C 90.000,E1 305.025} C_DIS
LIN {X 0.097,Y -672.673,Z 388.487,A 0.000,B 0.000,C 90.000,E1 303.579} C_DIS
LIN {X -0.034,Y -675.519,Z 388.481,A 0.000,B 0.000,C 90.000,E1 302.625} C_DIS
LIN {X 0.051,Y -678.909,Z 388.475,A 0.000,B 0.000,C 90.000,E1 301.416} C_DIS
LIN {X -0.006,Y -681.490,Z 388.469,A 0.000,B 0.000,C 90.000,E1 300.463} C_DIS
LIN {X -0.382,Y -683.815,Z 388.464,A 0.000,B 0.000,C 90.000,E1 299.539} C_DIS
LIN {X -0.131,Y -685.724,Z 388.459,A 0.000,B 0.000,C 90.000,E1 298.565} C_DIS
LIN {X 0.149,Y -687.303,Z 388.453,A 0.000,B 0.000,C 90.000,E1 297.590} C_DIS
LIN {X 0.061,Y -688.716,Z 388.447,A 0.000,B 0.000,C 90.000,E1 296.411} C_DIS
LIN {X -0.169,Y -689.461,Z 388.443,A 0.000,B 0.000,C 90.000,E1 295.720} C_DIS
LIN {X -0.389,Y -689.785,Z 388.439,A 0.000,B 0.000,C 90.000,E1 295.027} C_DIS
LIN {X -0.137,Y -689.800,Z 388.432,A 0.000,B 0.000,C 90.000,E1 293.823} C_DIS
LIN {X 0.049,Y -689.471,Z 388.430,A 0.000,B 0.000,C 90.000,E1 293.334} C_DIS
LIN {X 0.278,Y -689.445,Z 388.428,A 0.000,B 0.000,C 90.000,E1 293.078} C_DIS
LIN {X 0.055,Y -688.981,Z 388.424,A 0.000,B 0.000,C 90.000,E1 292.386} C_DIS
LIN {X 0.240,Y -688.588,Z 388.422,A 0.000,B 0.000,C 90.000,E1 291.897} C_DIS
LIN {X -0.035,Y -687.523,Z 388.417,A 0.000,B 0.000,C 90.000,E1 290.972} C_DIS
LIN {X 0.319,Y -686.219,Z 388.411,A 0.000,B 0.000,C 90.000,E1 289.993} C_DIS
LIN {X -0.191,Y -684.992,Z 388.407,A 0.000,B 0.000,C 90.000,E1 289.322} C_DIS
LIN {X -0.128,Y -682.856,Z 388.401,A 0.000,B 0.000,C 90.000,E1 288.127} C_DIS
LIN {X 0.112,Y -680.675,Z 388.394,A 0.000,B 0.000,C 90.000,E1 286.913} C_DIS
LIN {X 0.065,Y -677.905,Z 388.386,A 0.000,B 0.000,C 90.000,E1 285.481} C_DIS
LIN {X -0.161,Y -675.631,Z 388.379,A 0.000,B 0.000,C 90.000,E1 284.300} C_DIS
LIN {X -0.002,Y -671.659,Z 388.367,A 0.000,B 0.000,C 90.000,E1 282.119} C_DIS
LIN {X 0.112,Y -669.359,Z 388.359,A 0.000,B 0.000,C 90.000,E1 280.658} C_DIS
LIN {X 0.079,Y -665.830,Z 388.344,A 0.000,B 0.000,C 90.000,E1 277.992} C_DIS
LIN {X -0.043,Y -663.522,Z 388.331,A 0.000,B 0.000,C 90.000,E1 275.568} C_DIS
LIN {X 0.166,Y -661.949,Z 388.316,A 0.000,B 0.000,C 90.000,E1 272.865} C_DIS
LIN {X -0.084,Y -661.458,Z 388.304,A 0.000,B 0.000,C 90.000,E1 270.688} C_DIS
LIN {X -0.305,Y -661.242,Z 388.297,A 0.000,B 0.000,C 90.000,E1 269.484} C_DIS
LIN {X 0.126,Y -661.077,Z 388.290,A 0.000,B 0.000,C 90.000,E1 268.224} C_DIS
LIN {X 0.058,Y -660.959,Z 388.279,A 0.000,B 0.000,C 90.000,E1 266.274} C_DIS
LIN {X 0.022,Y -660.696,Z 388.274,A 0.000,B 0.000,C 90.000,E1 265.298} C_DIS
LIN {X 0.168,Y -660.219,Z 388.270,A 0.000,B 0.000,C 90.000,E1 264.552} C_DIS
LIN {X 0.054,Y -658.916,Z 388.263,A 0.000,B 0.000,C 90.000,E1 263.337} C_DIS
LIN {X -0.149,Y -658.552,Z 388.262,A 0.000,B 0.000,C 90.000,E1 263.109} C_DIS
LIN {X 0.176,Y -658.094,Z 388.259,A 0.000,B 0.000,C 90.000,E1 262.591} C_DIS
LIN {X 0.053,Y -657.686,Z 388.258,A 0.000,B 0.000,C 90.000,E1 262.356} C_DIS
LIN {X -0.157,Y -657.456,Z 388.256,A 0.000,B 0.000,C 90.000,E1 262.129} C_DIS
LIN {X -0.211,Y -655.281,Z 388.249,A 0.000,B 0.000,C 90.000,E1 260.905} C_DIS
LIN {X -0.038,Y -653.849,Z 388.245,A 0.000,B 0.000,C 90.000,E1 260.151} C_DIS
LIN {X -0.011,Y -651.766,Z 388.240,A 0.000,B 0.000,C 90.000,E1 259.162} C_DIS
LIN {X -0.016,Y -649.510,Z 388.234,A 0.000,B 0.000,C 90.000,E1 258.173} C_DIS
LIN {X 0.081,Y -647.109,Z 388.229,A 0.000,B 0.000,C 90.000,E1 257.173} C_DIS
LIN {X 0.291,Y -645.099,Z 388.225,A 0.000,B 0.000,C 90.000,E1 256.408} C_DIS
LIN {X -0.295,Y -642.291,Z 388.219,A 0.000,B 0.000,C 90.000,E1 255.463} C_DIS
LIN {X 0.324,Y -638.457,Z 388.212,A 0.000,B 0.000,C 90.000,E1 254.157} C_DIS
LIN {X 0.258,Y -634.200,Z 388.205,A 0.000,B 0.000,C 90.000,E1 252.906} C_DIS
LIN {X 0.308,Y -629.706,Z 388.198,A 0.000,B 0.000,C 90.000,E1 251.638} C_DIS
LIN {X -0.302,Y -625.812,Z 388.193,A 0.000,B 0.000,C 90.000,E1 250.678} C_DIS
LIN {X -0.183,Y -620.819,Z 388.185,A 0.000,B 0.000,C 90.000,E1 249.390} C_DIS
LIN {X -0.146,Y -615.670,Z 388.178,A 0.000,B 0.000,C 90.000,E1 248.103} C_DIS
LIN {X 0.033,Y -610.346,Z 388.171,A 0.000,B 0.000,C 90.000,E1 246.794} C_DIS
LIN {X 0.064,Y -603.724,Z 388.162,A 0.000,B 0.000,C 90.000,E1 245.229} C_DIS
LIN {X 0.284,Y -598.197,Z 388.155,A 0.000,B 0.000,C 90.000,E1 243.896} C_DIS
LIN {X -0.221,Y -591.536,Z 388.146,A 0.000,B 0.000,C 90.000,E1 242.359} C_DIS
LIN {X 0.095,Y -583.840,Z 388.136,A 0.000,B 0.000,C 90.000,E1 240.461} C_DIS
LIN {X 0.015,Y -576.430,Z 388.126,A 0.000,B 0.000,C 90.000,E1 238.584} C_DIS
LIN {X 0.009,Y -567.513,Z 388.112,A 0.000,B 0.000,C 90.000,E1 236.135} C_DIS
LIN {X 0.251,Y -560.049,Z 388.100,A 0.000,B 0.000,C 90.000,E1 233.909} C_DIS
LIN {X -0.251,Y -557.306,Z 388.095,A 0.000,B 0.000,C 90.000,E1 233.130} C_DIS
LIN {X 0.143,Y -552.567,Z 388.087,A 0.000,B 0.000,C 90.000,E1 231.698} C_DIS
LIN {X 0.009,Y -547.791,Z 388.080,A 0.000,B 0.000,C 90.000,E1 230.312} C_DIS
LIN {X 0.109,Y -542.126,Z 388.070,A 0.000,B 0.000,C 90.000,E1 228.609} C_DIS
LIN {X -0.264,Y -537.575,Z 388.062,A 0.000,B 0.000,C 90.000,E1 227.229} C_DIS
LIN {X -0.003,Y -532.242,Z 388.053,A 0.000,B 0.000,C 90.000,E1 225.486} C_DIS
LIN {X 0.078,Y -526.015,Z 388.042,A 0.000,B 0.000,C 90.000,E1 223.461} C_DIS
LIN {X 0.012,Y -520.015,Z 388.030,A 0.000,B 0.000,C 90.000,E1 221.434} C_DIS
LIN {X -0.233,Y -513.340,Z 388.017,A 0.000,B 0.000,C 90.000,E1 219.116} C_DIS
LIN {X 0.088,Y -509.351,Z 388.009,A 0.000,B 0.000,C 90.000,E1 217.604} C_DIS
LIN {X 0.021,Y -503.185,Z 387.996,A 0.000,B 0.000,C 90.000,E1 215.231} C_DIS
LIN {X 0.134,Y -498.689,Z 387.986,A 0.000,B 0.000,C 90.000,E1 213.420} C_DIS
LIN {X 0.015,Y -495.150,Z 387.977,A 0.000,B 0.000,C 90.000,E1 211.926} C_DIS
LIN {X -0.165,Y -490.940,Z 387.967,A 0.000,B 0.000,C 90.000,E1 210.129} C_DIS
LIN {X -0.011,Y -486.059,Z 387.955,A 0.000,B 0.000,C 90.000,E1 207.975} C_DIS
LIN {X 0.224,Y -481.709,Z 387.945,A 0.000,B 0.000,C 90.000,E1 206.104} C_DIS
LIN {X 0.140,Y -477.338,Z 387.935,A 0.000,B 0.000,C 90.000,E1 204.259} C_DIS
LIN {X 0.035,Y -473.529,Z 387.926,A 0.000,B 0.000,C 90.000,E1 202.717} C_DIS
LIN {X -0.003,Y -469.058,Z 387.916,A 0.000,B 0.000,C 90.000,E1 200.844} C_DIS
LIN {X -0.115,Y -463.980,Z 387.904,A 0.000,B 0.000,C 90.000,E1 198.652} C_DIS
LIN {X -0.203,Y -459.315,Z 387.891,A 0.000,B 0.000,C 90.000,E1 196.441} C_DIS
LIN {X -0.207,Y -454.327,Z 387.877,A 0.000,B 0.000,C 90.000,E1 193.883} C_DIS
LIN {X 0.096,Y -450.213,Z 387.865,A 0.000,B 0.000,C 90.000,E1 191.591} C_DIS
LIN {X -0.077,Y -446.940,Z 387.854,A 0.000,B 0.000,C 90.000,E1 189.670} C_DIS
LIN {X 0.215,Y -443.412,Z 387.841,A 0.000,B 0.000,C 90.000,E1 187.352} C_DIS
LIN {X 0.010,Y -439.734,Z 387.827,A 0.000,B 0.000,C 90.000,E1 184.759} C_DIS
LIN {X 0.038,Y -436.745,Z 387.812,A 0.000,B 0.000,C 90.000,E1 182.121} C_DIS
LIN {X -0.186,Y -433.765,Z 387.792,A 0.000,B 0.000,C 90.000,E1 178.511} C_DIS
LIN {X 0.146,Y -431.989,Z 387.768,A 0.000,B 0.000,C 90.000,E1 174.147} C_DIS
LIN {X -0.104,Y -432.325,Z 387.736,A 0.000,B 0.000,C 90.000,E1 168.522} C_DIS
LIN {X -0.008,Y -435.793,Z 387.707,A 0.000,B 0.000,C 90.000,E1 163.196} C_DIS
LIN {X 0.201,Y -440.214,Z 387.685,A 0.000,B 0.000,C 90.000,E1 159.209} C_DIS
LIN {X 0.056,Y -446.616,Z 387.661,A 0.000,B 0.000,C 90.000,E1 154.973} C_DIS
LIN {X -0.072,Y -454.014,Z 387.639,A 0.000,B 0.000,C 90.000,E1 151.101} C_DIS
LIN {X 0.036,Y -463.230,Z 387.618,A 0.000,B 0.000,C 90.000,E1 147.248} C_DIS
LIN {X -0.012,Y -473.376,Z 387.599,A 0.000,B 0.000,C 90.000,E1 143.783} C_DIS
LIN {X -0.034,Y -481.470,Z 387.585,A 0.000,B 0.000,C 90.000,E1 141.295} C_DIS
LIN {X 0.028,Y -486.646,Z 387.576,A 0.000,B 0.000,C 90.000,E1 139.747} C_DIS
LIN {X -0.192,Y -491.789,Z 387.568,A 0.000,B 0.000,C 90.000,E1 138.243} C_DIS
LIN {X 0.161,Y -495.678,Z 387.561,A 0.000,B 0.000,C 90.000,E1 136.986} C_DIS
LIN {X -0.127,Y -499.334,Z 387.554,A 0.000,B 0.000,C 90.000,E1 135.810} C_DIS
LIN {X -0.016,Y -502.749,Z 387.548,A 0.000,B 0.000,C 90.000,E1 134.595} C_DIS
LIN {X -0.078,Y -505.039,Z 387.543,A 0.000,B 0.000,C 90.000,E1 133.704} C_DIS
LIN {X 0.251,Y -507.116,Z 387.538,A 0.000,B 0.000,C 90.000,E1 132.771} C_DIS
LIN {X -0.110,Y -508.987,Z 387.533,A 0.000,B 0.000,C 90.000,E1 131.919} C_DIS
LIN {X 0.265,Y -510.579,Z 387.528,A 0.000,B 0.000,C 90.000,E1 130.987} C_DIS
LIN {X 0.322,Y -511.966,Z 387.523,A 0.000,B 0.000,C 90.000,E1 130.092} C_DIS
LIN {X -0.325,Y -512.990,Z 387.518,A 0.000,B 0.000,C 90.000,E1 129.277} C_DIS
LIN {X -0.241,Y -513.658,Z 387.513,A 0.000,B 0.000,C 90.000,E1 128.382} C_DIS
LIN {X 0.252,Y -513.706,Z 387.508,A 0.000,B 0.000,C 90.000,E1 127.443} C_DIS
LIN {X 0.026,Y -513.243,Z 387.503,A 0.000,B 0.000,C 90.000,E1 126.583} C_DIS
LIN {X -0.205,Y -512.407,Z 387.498,A 0.000,B 0.000,C 90.000,E1 125.724} C_DIS
LIN {X -0.029,Y -511.250,Z 387.493,A 0.000,B 0.000,C 90.000,E1 124.818} C_DIS
LIN {X 0.221,Y -510.291,Z 387.490,A 0.000,B 0.000,C 90.000,E1 124.199} C_DIS
LIN {X -0.333,Y -508.478,Z 387.485,A 0.000,B 0.000,C 90.000,E1 123.372} C_DIS
LIN {X 0.222,Y -506.264,Z 387.480,A 0.000,B 0.000,C 90.000,E1 122.418} C_DIS
LIN {X 0.054,Y -503.720,Z 387.475,A 0.000,B 0.000,C 90.000,E1 121.544} C_DIS
LIN {X 0.242,Y -501.836,Z 387.472,A 0.000,B 0.000,C 90.000,E1 120.924} C_DIS
LIN {X 0.021,Y -498.727,Z 387.467,A 0.000,B 0.000,C 90.000,E1 120.050} C_DIS
LIN {X -0.006,Y -494.718,Z 387.461,A 0.000,B 0.000,C 90.000,E1 118.999} C_DIS
LIN {X 0.089,Y -491.585,Z 387.457,A 0.000,B 0.000,C 90.000,E1 118.231} C_DIS
LIN {X -0.041,Y -486.987,Z 387.451,A 0.000,B 0.000,C 90.000,E1 117.180} C_DIS
LIN {X -0.238,Y -481.274,Z 387.444,A 0.000,B 0.000,C 90.000,E1 115.976} C_DIS
LIN {X -0.109,Y -474.637,Z 387.436,A 0.000,B 0.000,C 90.000,E1 114.567} C_DIS
LIN {X -0.206,Y -469.978,Z 387.431,A 0.000,B 0.000,C 90.000,E1 113.643} C_DIS
LIN {X 0.203,Y -463.693,Z 387.424,A 0.000,B 0.000,C 90.000,E1 112.333} C_DIS
LIN {X 0.077,Y -456.550,Z 387.416,A 0.000,B 0.000,C 90.000,E1 110.918} C_DIS
LIN {X 0.065,Y -455.016,Z 387.415,A 0.000,B 0.000,C 90.000,E1 110.610} C_DIS
LIN {X 0.025,Y -455.019,Z 387.415,A 0.000,B 0.000,C 90.000,E1 110.610} C_DIS
LIN {X -0.049,Y -457.260,Z 387.410,A 0.000,B 0.000,C 90.000,E1 109.812} C_DIS
LIN {X 0.020,Y -465.881,Z 387.387,A 0.000,B 0.000,C 90.000,E1 105.662} C_DIS
LIN {X 0.190,Y -467.442,Z 387.384,A 0.000,B 0.000,C 90.000,E1 105.009} C_DIS
LIN {X -0.004,Y -468.058,Z 387.382,A 0.000,B 0.000,C 90.000,E1 104.717} C_DIS
LIN {X 0.135,Y -475.698,Z 387.357,A 0.000,B 0.000,C 90.000,E1 100.310} C_DIS
LIN {X -0.028,Y -476.260,Z 387.356,A 0.000,B 0.000,C 90.000,E1 100.018} C_DIS
LIN {X 0.237,Y -482.148,Z 387.330,A 0.000,B 0.000,C 90.000,E1 95.334} C_DIS
LIN {X -0.008,Y -485.536,Z 387.304,A 0.000,B 0.000,C 90.000,E1 90.745} C_DIS
LIN {X 0.025,Y -486.377,Z 387.280,A 0.000,B 0.000,C 90.000,E1 86.445} C_DIS
LIN {X -0.152,Y -486.338,Z 387.279,A 0.000,B 0.000,C 90.000,E1 86.159} C_DIS
LIN {X -0.073,Y -484.648,Z 387.253,A 0.000,B 0.000,C 90.000,E1 81.546} C_DIS
LIN {X -0.182,Y -480.570,Z 387.227,A 0.000,B 0.000,C 90.000,E1 76.937} C_DIS
LIN {X 0.097,Y -477.729,Z 387.217,A 0.000,B 0.000,C 90.000,E1 75.046} C_DIS
LIN {X 0.017,Y -473.950,Z 387.200,A 0.000,B 0.000,C 90.000,E1 71.945} C_DIS
LIN {X 0.231,Y -473.000,Z 387.197,A 0.000,B 0.000,C 90.000,E1 71.456} C_DIS
LIN {X 0.190,Y -473.033,Z 387.197,A 0.000,B 0.000,C 90.000,E1 71.456} C_DIS
LIN {X -0.068,Y -482.010,Z 387.190,A 0.000,B 0.000,C 90.000,E1 70.242} C_DIS
LIN {X -0.047,Y -492.978,Z 387.182,A 0.000,B 0.000,C 90.000,E1 68.720} C_DIS
LIN {X -0.220,Y -496.166,Z 387.179,A 0.000,B 0.000,C 90.000,E1 68.284} C_DIS
LIN {X -0.239,Y -503.313,Z 387.173,A 0.000,B 0.000,C 90.000,E1 67.230} C_DIS
LIN {X -0.038,Y -507.968,Z 387.169,A 0.000,B 0.000,C 90.000,E1 66.485} C_DIS
LIN {X 0.160,Y -511.578,Z 387.166,A 0.000,B 0.000,C 90.000,E1 65.869} C_DIS
LIN {X -0.044,Y -515.603,Z 387.162,A 0.000,B 0.000,C 90.000,E1 65.153} C_DIS
LIN {X 0.209,Y -518.571,Z 387.159,A 0.000,B 0.000,C 90.000,E1 64.537} C_DIS
LIN {X 0.012,Y -521.319,Z 387.155,A 0.000,B 0.000,C 90.000,E1 63.973} C_DIS
LIN {X 0.223,Y -523.266,Z 387.153,A 0.000,B 0.000,C 90.000,E1 63.512} C_DIS
LIN {X -0.022,Y -526.680,Z 387.148,A 0.000,B 0.000,C 90.000,E1 62.666} C_DIS
LIN {X -0.128,Y -528.859,Z 387.145,A 0.000,B 0.000,C 90.000,E1 62.103} C_DIS
LIN {X -0.020,Y -530.923,Z 387.142,A 0.000,B 0.000,C 90.000,E1 61.513} C_DIS
LIN {X -0.063,Y -531.763,Z 387.140,A 0.000,B 0.000,C 90.000,E1 61.229} C_DIS
LIN {X 0.107,Y -532.785,Z 387.139,A 0.000,B 0.000,C 90.000,E1 60.923} C_DIS
LIN {X -0.042,Y -535.334,Z 387.134,A 0.000,B 0.000,C 90.000,E1 60.078} C_DIS
LIN {X 0.104,Y -537.677,Z 387.129,A 0.000,B 0.000,C 90.000,E1 59.203} C_DIS
LIN {X 0.281,Y -539.867,Z 387.124,A 0.000,B 0.000,C 90.000,E1 58.329} C_DIS
LIN {X 0.025,Y -541.855,Z 387.120,A 0.000,B 0.000,C 90.000,E1 57.502} C_DIS
LIN {X -0.027,Y -544.029,Z 387.113,A 0.000,B 0.000,C 90.000,E1 56.373} C_DIS
LIN {X 0.065,Y -545.353,Z 387.109,A 0.000,B 0.000,C 90.000,E1 55.515} C_DIS
LIN {X -0.133,Y -546.378,Z 387.104,A 0.000,B 0.000,C 90.000,E1 54.689} C_DIS
LIN {X -0.049,Y -546.917,Z 387.101,A 0.000,B 0.000,C 90.000,E1 54.116} C_DIS
LIN {X 0.134,Y -547.443,Z 387.094,A 0.000,B 0.000,C 90.000,E1 52.970} C_DIS
LIN {X -0.059,Y -547.598,Z 387.090,A 0.000,B 0.000,C 90.000,E1 52.145} C_DIS
LIN {X -0.011,Y -547.416,Z 387.085,A 0.000,B 0.000,C 90.000,E1 51.295} C_DIS
LIN {X 0.123,Y -546.935,Z 387.080,A 0.000,B 0.000,C 90.000,E1 50.436} C_DIS
LIN {X -0.175,Y -546.142,Z 387.076,A 0.000,B 0.000,C 90.000,E1 49.622} C_DIS
LIN {X -0.126,Y -545.158,Z 387.071,A 0.000,B 0.000,C 90.000,E1 48.771} C_DIS
LIN {X -0.058,Y -543.548,Z 387.065,A 0.000,B 0.000,C 90.000,E1 47.634} C_DIS
LIN {X 0.345,Y -541.010,Z 387.055,A 0.000,B 0.000,C 90.000,E1 45.891} C_DIS
LIN {X 0.279,Y -537.665,Z 387.043,A 0.000,B 0.000,C 90.000,E1 43.623} C_DIS
LIN {X 0.188,Y -535.375,Z 387.033,A 0.000,B 0.000,C 90.000,E1 41.919} C_DIS
LIN {X 0.033,Y -532.833,Z 387.022,A 0.000,B 0.000,C 90.000,E1 39.930} C_DIS
LIN {X 0.318,Y -530.958,Z 387.014,A 0.000,B 0.000,C 90.000,E1 38.463} C_DIS
LIN {X -0.176,Y -529.119,Z 387.006,A 0.000,B 0.000,C 90.000,E1 37.076} C_DIS
LIN {X 0.116,Y -526.838,Z 386.996,A 0.000,B 0.000,C 90.000,E1 35.311} C_DIS
LIN {X 0.019,Y -524.171,Z 386.985,A 0.000,B 0.000,C 90.000,E1 33.293} C_DIS
LIN {X 0.000,Y -521.501,Z 386.974,A 0.000,B 0.000,C 90.000,E1 31.258} C_DIS
LIN {X -0.288,Y -519.265,Z 386.964,A 0.000,B 0.000,C 90.000,E1 29.539} C_DIS
LIN {X -0.047,Y -516.801,Z 386.953,A 0.000,B 0.000,C 90.000,E1 27.462} C_DIS
LIN {X -0.104,Y -514.516,Z 386.941,A 0.000,B 0.000,C 90.000,E1 25.412} C_DIS
LIN {X 0.024,Y -512.397,Z 386.930,A 0.000,B 0.000,C 90.000,E1 23.334} C_DIS
LIN {X -0.225,Y -510.779,Z 386.920,A 0.000,B 0.000,C 90.000,E1 21.589} C_DIS
LIN {X -0.189,Y -508.959,Z 386.907,A 0.000,B 0.000,C 90.000,E1 19.214} C_DIS
LIN {X 0.177,Y -507.587,Z 386.895,A 0.000,B 0.000,C 90.000,E1 17.094} C_DIS
LIN {X 0.201,Y -506.490,Z 386.884,A 0.000,B 0.000,C 90.000,E1 15.009} C_DIS
LIN {X 0.009,Y -505.554,Z 386.870,A 0.000,B 0.000,C 90.000,E1 12.647} C_DIS
LIN {X -0.045,Y -505.051,Z 386.854,A 0.000,B 0.000,C 90.000,E1 9.670} C_DIS
LIN {X 0.274,Y -505.262,Z 386.839,A 0.000,B 0.000,C 90.000,E1 6.947} C_DIS
LIN {X -0.069,Y -506.128,Z 386.824,A 0.000,B 0.000,C 90.000,E1 4.302} C_DIS
LIN {X -0.007,Y -508.057,Z 386.807,A 0.000,B 0.000,C 90.000,E1 1.318} C_DIS
LIN {X 0.184,Y -511.424,Z 386.789,A 0.000,B 0.000,C 90.000,E1 357.993} C_DIS
LIN {X -0.211,Y -513.395,Z 386.781,A 0.000,B 0.000,C 90.000,E1 356.560} C_DIS
LIN {X -0.218,Y -516.973,Z 386.768,A 0.000,B 0.000,C 90.000,E1 354.204} C_DIS
LIN {X -0.017,Y -521.670,Z 386.753,A 0.000,B 0.000,C 90.000,E1 351.546} C_DIS
LIN {X 0.107,Y -529.871,Z 386.732,A 0.000,B 0.000,C 90.000,E1 347.757} C_DIS
LIN {X 0.040,Y -535.857,Z 386.719,A 0.000,B 0.000,C 90.000,E1 345.463} C_DIS
LIN {X 0.198,Y -541.357,Z 386.708,A 0.000,B 0.000,C 90.000,E1 343.449} C_DIS
LIN {X -0.023,Y -545.332,Z 386.700,A 0.000,B 0.000,C 90.000,E1 342.054} C_DIS
LIN {X -0.086,Y -550.194,Z 386.691,A 0.000,B 0.000,C 90.000,E1 340.369} C_DIS
LIN {X 0.047,Y -554.277,Z 386.683,A 0.000,B 0.000,C 90.000,E1 338.954} C_DIS
LIN {X 0.043,Y -559.275,Z 386.674,A 0.000,B 0.000,C 90.000,E1 337.283} C_DIS
LIN {X -0.057,Y -565.085,Z 386.663,A 0.000,B 0.000,C 90.000,E1 335.357} C_DIS
LIN {X -0.135,Y -570.155,Z 386.654,A 0.000,B 0.000,C 90.000,E1 333.717} C_DIS
LIN {X -0.100,Y -575.332,Z 386.645,A 0.000,B 0.000,C 90.000,E1 332.076} C_DIS
LIN {X -0.071,Y -579.862,Z 386.637,A 0.000,B 0.000,C 90.000,E1 330.717} C_DIS
LIN {X 0.047,Y -586.203,Z 386.627,A 0.000,B 0.000,C 90.000,E1 328.820} C_DIS
LIN {X -0.153,Y -590.670,Z 386.619,A 0.000,B 0.000,C 90.000,E1 327.502} C_DIS
LIN {X -0.258,Y -597.929,Z 386.608,A 0.000,B 0.000,C 90.000,E1 325.388} C_DIS
LIN {X 0.105,Y -602.563,Z 386.600,A 0.000,B 0.000,C 90.000,E1 324.036} C_DIS
LIN {X 0.249,Y -609.152,Z 386.590,A 0.000,B 0.000,C 90.000,E1 322.190} C_DIS
LIN {X -0.037,Y -615.844,Z 386.580,A 0.000,B 0.000,C 90.000,E1 320.400} C_DIS
LIN {X 0.145,Y -620.667,Z 386.573,A 0.000,B 0.000,C 90.000,E1 319.094} C_DIS
LIN {X 0.197,Y -626.282,Z 386.564,A 0.000,B 0.000,C 90.000,E1 317.553} C_DIS
LIN {X 0.141,Y -629.960,Z 386.559,A 0.000,B 0.000,C 90.000,E1 316.539} C_DIS
LIN {X -0.325,Y -633.574,Z 386.553,A 0.000,B 0.000,C 90.000,E1 315.567} C_DIS
LIN {X 0.063,Y -638.169,Z 386.546,A 0.000,B 0.000,C 90.000,E1 314.271} C_DIS
LIN {X 0.169,Y -641.868,Z 386.540,A 0.000,B 0.000,C 90.000,E1 313.257} C_DIS
LIN {X -0.148,Y -645.622,Z 386.535,A 0.000,B 0.000,C 90.000,E1 312.285} C_DIS
LIN {X -0.074,Y -652.031,Z 386.525,A 0.000,B 0.000,C 90.000,E1 310.539} C_DIS
LIN {X 0.189,Y -657.288,Z 386.517,A 0.000,B 0.000,C 90.000,E1 309.036} C_DIS
LIN {X 0.177,Y -661.413,Z 386.510,A 0.000,B 0.000,C 90.000,E1 307.810} C_DIS
LIN {X 0.218,Y -663.074,Z 386.507,A 0.000,B 0.000,C 90.000,E1 307.317} C_DIS
LIN {X -0.122,Y -667.710,Z 386.499,A 0.000,B 0.000,C 90.000,E1 305.884} C_DIS
LIN {X 0.060,Y -670.645,Z 386.494,A 0.000,B 0.000,C 90.000,E1 304.898} C_DIS
LIN {X 0.025,Y -674.967,Z 386.486,A 0.000,B 0.000,C 90.000,E1 303.452} C_DIS
LIN {X -0.246,Y -677.070,Z 386.482,A 0.000,B 0.000,C 90.000,E1 302.752} C_DIS
LIN {X -0.109,Y -678.338,Z 386.479,A 0.000,B 0.000,C 90.000,E1 302.260} C_DIS
LIN {X 0.069,Y -679.102,Z 386.478,A 0.000,B 0.000,C 90.000,E1 302.005} C_DIS
LIN {X -0.140,Y -680.309,Z 386.475,A 0.000,B 0.000,C 90.000,E1 301.544} C_DIS
LIN {X 0.404,Y -681.073,Z 386.474,A 0.000,B 0.000,C 90.000,E1 301.258} C_DIS
LIN {X 0.208,Y -682.207,Z 386.471,A 0.000,B 0.000,C 90.000,E1 300.797} C_DIS
LIN {X -0.181,Y -682.980,Z 386.470,A 0.000,B 0.000,C 90.000,E1 300.590} C_DIS
LIN {X 0.226,Y -683.975,Z 386.467,A 0.000,B 0.000,C 90.000,E1 300.079} C_DIS
LIN {X 0.053,Y -685.130,Z 386.465,A 0.000,B 0.000,C 90.000,E1 299.617} C_DIS
LIN {X 0.105,Y -686.540,Z 386.461,A 0.000,B 0.000,C 90.000,E1 298.899} C_DIS
LIN {X 0.019,Y -688.354,Z 386.454,A 0.000,B 0.000,C 90.000,E1 297.719} C_DIS
LIN {X 0.098,Y -689.110,Z 386.450,A 0.000,B 0.000,C 90.000,E1 297.001} C_DIS
LIN {X -0.276,Y -690.167,Z 386.444,A 0.000,B 0.000,C 90.000,E1 295.848} C_DIS
LIN {X 0.137,Y -690.535,Z 386.440,A 0.000,B 0.000,C 90.000,E1 295.103} C_DIS
LIN {X 0.172,Y -690.410,Z 386.434,A 0.000,B 0.000,C 90.000,E1 294.155} C_DIS
LIN {X 0.010,Y -690.181,Z 386.432,A 0.000,B 0.000,C 90.000,E1 293.695} C_DIS
LIN {X -0.246,Y -689.430,Z 386.426,A 0.000,B 0.000,C 90.000,E1 292.770} C_DIS
LIN {X 0.168,Y -688.680,Z 386.422,A 0.000,B 0.000,C 90.000,E1 292.025} C_DIS
LIN {X -0.285,Y -687.887,Z 386.420,A 0.000,B 0.000,C 90.000,E1 291.589} C_DIS
LIN {X -0.136,Y -687.068,Z 386.416,A 0.000,B 0.000,C 90.000,E1 290.865} C_DIS
LIN {X 0.218,Y -685.544,Z 386.411,A 0.000,B 0.000,C 90.000,E1 289.885} C_DIS
LIN {X -0.167,Y -682.942,Z 386.403,A 0.000,B 0.000,C 90.000,E1 288.489} C_DIS
LIN {X 0.043,Y -680.303,Z 386.395,A 0.000,B 0.000,C 90.000,E1 287.040} C_DIS
LIN {X -0.049,Y -676.960,Z 386.385,A 0.000,B 0.000,C 90.000,E1 285.371} C_DIS
LIN {X -0.117,Y -674.588,Z 386.379,A 0.000,B 0.000,C 90.000,E1 284.175} C_DIS
LIN {X 0.308,Y -669.464,Z 386.363,A 0.000,B 0.000,C 90.000,E1 281.243} C_DIS
LIN {X -0.191,Y -665.923,Z 386.349,A 0.000,B 0.000,C 90.000,E1 278.859} C_DIS
LIN {X -0.065,Y -662.733,Z 386.332,A 0.000,B 0.000,C 90.000,E1 275.682} C_DIS
LIN {X 0.111,Y -661.120,Z 386.317,A 0.000,B 0.000,C 90.000,E1 272.980} C_DIS
LIN {X 0.316,Y -660.597,Z 386.303,A 0.000,B 0.000,C 90.000,E1 270.516} C_DIS
LIN {X -0.279,Y -660.494,Z 386.294,A 0.000,B 0.000,C 90.000,E1 268.854} C_DIS
LIN {X -0.207,Y -660.337,Z 386.284,A 0.000,B 0.000,C 90.000,E1 267.135} C_DIS
LIN {X -0.248,Y -660.379,Z 386.279,A 0.000,B 0.000,C 90.000,E1 266.159} C_DIS
LIN {X -0.238,Y -660.148,Z 386.273,A 0.000,B 0.000,C 90.000,E1 265.179} C_DIS
LIN {X 0.244,Y -659.380,Z 386.266,A 0.000,B 0.000,C 90.000,E1 263.913} C_DIS
LIN {X -0.077,Y -659.010,Z 386.264,A 0.000,B 0.000,C 90.000,E1 263.451} C_DIS
LIN {X -0.277,Y -658.699,Z 386.262,A 0.000,B 0.000,C 90.000,E1 263.223} C_DIS
LIN {X 0.049,Y -658.343,Z 386.260,A 0.000,B 0.000,C 90.000,E1 262.704} C_DIS
LIN {X 0.249,Y -657.575,Z 386.255,A 0.000,B 0.000,C 90.000,E1 261.951} C_DIS
LIN {X -0.206,Y -656.480,Z 386.251,A 0.000,B 0.000,C 90.000,E1 261.254} C_DIS
LIN {X 0.271,Y -654.233,Z 386.245,A 0.000,B 0.000,C 90.000,E1 259.982} C_DIS
LIN {X -0.217,Y -652.721,Z 386.240,A 0.000,B 0.000,C 90.000,E1 259.285} C_DIS
LIN {X -0.082,Y -650.582,Z 386.235,A 0.000,B 0.000,C 90.000,E1 258.285} C_DIS
LIN {X -0.246,Y -647.699,Z 386.228,A 0.000,B 0.000,C 90.000,E1 257.061} C_DIS
LIN {X -0.033,Y -645.773,Z 386.224,A 0.000,B 0.000,C 90.000,E1 256.297} C_DIS
LIN {X 0.171,Y -643.050,Z 386.218,A 0.000,B 0.000,C 90.000,E1 255.283} C_DIS
LIN {X 0.174,Y -640.053,Z 386.213,A 0.000,B 0.000,C 90.000,E1 254.283} C_DIS
LIN {X -0.138,Y -637.591,Z 386.209,A 0.000,B 0.000,C 90.000,E1 253.559} C_DIS
LIN {X 0.142,Y -635.068,Z 386.204,A 0.000,B 0.000,C 90.000,E1 252.779} C_DIS
LIN {X 0.206,Y -631.500,Z 386.199,A 0.000,B 0.000,C 90.000,E1 251.764} C_DIS
LIN {X -0.181,Y -628.711,Z 386.195,A 0.000,B 0.000,C 90.000,E1 251.040} C_DIS
LIN {X -0.013,Y -623.759,Z 386.188,A 0.000,B 0.000,C 90.000,E1 249.752} C_DIS
LIN {X 0.077,Y -618.680,Z 386.180,A 0.000,B 0.000,C 90.000,E1 248.465} C_DIS
LIN {X 0.072,Y -613.398,Z 386.173,A 0.000,B 0.000,C 90.000,E1 247.177} C_DIS
LIN {X -0.308,Y -609.045,Z 386.168,A 0.000,B 0.000,C 90.000,E1 246.177} C_DIS
LIN {X 0.006,Y -603.545,Z 386.160,A 0.000,B 0.000,C 90.000,E1 244.845} C_DIS
LIN {X 0.225,Y -598.010,Z 386.153,A 0.000,B 0.000,C 90.000,E1 243.512} C_DIS
LIN {X -0.284,Y -591.379,Z 386.144,A 0.000,B 0.000,C 90.000,E1 241.975} C_DIS
LIN {X 0.058,Y -581.623,Z 386.131,A 0.000,B 0.000,C 90.000,E1 239.537} C_DIS
LIN {X 0.028,Y -571.450,Z 386.116,A 0.000,B 0.000,C 90.000,E1 236.834} C_DIS
LIN {X 0.054,Y -563.886,Z 386.104,A 0.000,B 0.000,C 90.000,E1 234.642} C_DIS
LIN {X 0.117,Y -559.343,Z 386.096,A 0.000,B 0.000,C 90.000,E1 233.256} C_DIS
LIN {X -0.227,Y -554.617,Z 386.088,A 0.000,B 0.000,C 90.000,E1 231.904} C_DIS
LIN {X 0.033,Y -549.844,Z 386.081,A 0.000,B 0.000,C 90.000,E1 230.481} C_DIS
LIN {X -0.133,Y -543.239,Z 386.070,A 0.000,B 0.000,C 90.000,E1 228.528} C_DIS
LIN {X -0.113,Y -537.790,Z 386.060,A 0.000,B 0.000,C 90.000,E1 226.824} C_DIS
LIN {X -0.197,Y -533.330,Z 386.052,A 0.000,B 0.000,C 90.000,E1 225.405} C_DIS
LIN {X -0.028,Y -528.010,Z 386.043,A 0.000,B 0.000,C 90.000,E1 223.662} C_DIS
LIN {X -0.026,Y -521.950,Z 386.031,A 0.000,B 0.000,C 90.000,E1 221.634} C_DIS
LIN {X 0.130,Y -515.237,Z 386.018,A 0.000,B 0.000,C 90.000,E1 219.277} C_DIS
LIN {X 0.084,Y -511.238,Z 386.010,A 0.000,B 0.000,C 90.000,E1 217.810} C_DIS
LIN {X 0.069,Y -504.996,Z 385.997,A 0.000,B 0.000,C 90.000,E1 215.438} C_DIS
LIN {X 0.343,Y -501.257,Z 385.989,A 0.000,B 0.000,C 90.000,E1 213.913} C_DIS
LIN {X 0.136,Y -496.963,Z 385.979,A 0.000,B 0.000,C 90.000,E1 212.133} C_DIS
LIN {X 0.260,Y -492.037,Z 385.967,A 0.000,B 0.000,C 90.000,E1 210.001} C_DIS
LIN {X -0.229,Y -487.849,Z 385.957,A 0.000,B 0.000,C 90.000,E1 208.231} C_DIS
LIN {X 0.050,Y -483.582,Z 385.947,A 0.000,B 0.000,C 90.000,E1 206.360} C_DIS
LIN {X 0.011,Y -479.201,Z 385.936,A 0.000,B 0.000,C 90.000,E1 204.515} C_DIS
LIN {X 0.128,Y -475.432,Z 385.928,A 0.000,B 0.000,C 90.000,E1 202.950} C_DIS
LIN {X -0.008,Y -471.681,Z 385.919,A 0.000,B 0.000,C 90.000,E1 201.408} C_DIS
LIN {X 0.015,Y -467.278,Z 385.909,A 0.000,B 0.000,C 90.000,E1 199.523} C_DIS
LIN {X 0.090,Y -461.795,Z 385.894,A 0.000,B 0.000,C 90.000,E1 196.985} C_DIS
LIN {X -0.170,Y -455.510,Z 385.877,A 0.000,B 0.000,C 90.000,E1 193.828} C_DIS
LIN {X -0.034,Y -451.954,Z 385.866,A 0.000,B 0.000,C 90.000,E1 191.883} C_DIS
LIN {X 0.024,Y -448.108,Z 385.853,A 0.000,B 0.000,C 90.000,E1 189.613} C_DIS
LIN {X 0.176,Y -445.036,Z 385.843,A 0.000,B 0.000,C 90.000,E1 187.644} C_DIS
LIN {X -0.084,Y -441.744,Z 385.830,A 0.000,B 0.000,C 90.000,E1 185.391} C_DIS
LIN {X 0.137,Y -438.175,Z 385.814,A 0.000,B 0.000,C 90.000,E1 182.407} C_DIS
LIN {X -0.029,Y -435.060,Z 385.793,A 0.000,B 0.000,C 90.000,E1 178.797} C_DIS
LIN {X -0.018,Y -433.491,Z 385.777,A 0.000,B 0.000,C 90.000,E1 175.812} C_DIS
LIN {X -0.220,Y -432.851,Z 385.764,A 0.000,B 0.000,C 90.000,E1 173.514} C_DIS
LIN {X 0.142,Y -433.232,Z 385.738,A 0.000,B 0.000,C 90.000,E1 168.814} C_DIS
LIN {X 0.179,Y -436.462,Z 385.709,A 0.000,B 0.000,C 90.000,E1 163.504} C_DIS
LIN {X -0.198,Y -439.196,Z 385.694,A 0.000,B 0.000,C 90.000,E1 160.913} C_DIS
LIN {X 0.071,Y -442.955,Z 385.677,A 0.000,B 0.000,C 90.000,E1 157.922} C_DIS
LIN {X 0.030,Y -448.170,Z 385.659,A 0.000,B 0.000,C 90.000,E1 154.665} C_DIS
LIN {X 0.065,Y -456.427,Z 385.636,A 0.000,B 0.000,C 90.000,E1 150.461} C_DIS
LIN {X 0.131,Y -466.000,Z 385.615,A 0.000,B 0.000,C 90.000,E1 146.628} C_DIS
LIN {X 0.030,Y -475.435,Z 385.597,A 0.000,B 0.000,C 90.000,E1 143.497} C_DIS
LIN {X -0.040,Y -482.569,Z 385.585,A 0.000,B 0.000,C 90.000,E1 141.331} C_DIS
LIN {X 0.210,Y -486.730,Z 385.578,A 0.000,B 0.000,C 90.000,E1 140.070} C_DIS
LIN {X -0.011,Y -491.882,Z 385.570,A 0.000,B 0.000,C 90.000,E1 138.566} C_DIS
LIN {X 0.162,Y -494.907,Z 385.565,A 0.000,B 0.000,C 90.000,E1 137.634} C_DIS
LIN {X -0.140,Y -498.660,Z 385.558,A 0.000,B 0.000,C 90.000,E1 136.458} C_DIS
LIN {X -0.041,Y -502.170,Z 385.551,A 0.000,B 0.000,C 90.000,E1 135.243} C_DIS
LIN {X -0.107,Y -504.654,Z 385.546,A 0.000,B 0.000,C 90.000,E1 134.352} C_DIS
LIN {X -0.150,Y -506.846,Z 385.541,A 0.000,B 0.000,C 90.000,E1 133.461} C_DIS
LIN {X 0.200,Y -508.820,Z 385.536,A 0.000,B 0.000,C 90.000,E1 132.528} C_DIS
LIN {X -0.146,Y -510.576,Z 385.531,A 0.000,B 0.000,C 90.000,E1 131.676} C_DIS
LIN {X -0.089,Y -512.110,Z 385.527,A 0.000,B 0.000,C 90.000,E1 130.782} C_DIS
LIN {X 0.072,Y -513.019,Z 385.523,A 0.000,B 0.000,C 90.000,E1 130.172} C_DIS
LIN {X 0.158,Y -514.043,Z 385.518,A 0.000,B 0.000,C 90.000,E1 129.277} C_DIS
LIN {X 0.008,Y -514.517,Z 385.515,A 0.000,B 0.000,C 90.000,E1 128.705} C_DIS
LIN {X 0.182,Y -514.718,Z 385.512,A 0.000,B 0.000,C 90.000,E1 128.096} C_DIS
LIN {X -0.032,Y -514.638,Z 385.507,A 0.000,B 0.000,C 90.000,E1 127.237} C_DIS
LIN {X -0.247,Y -514.040,Z 385.502,A 0.000,B 0.000,C 90.000,E1 126.377} C_DIS
LIN {X -0.050,Y -513.116,Z 385.497,A 0.000,B 0.000,C 90.000,E1 125.471} C_DIS
LIN {X -0.282,Y -511.874,Z 385.492,A 0.000,B 0.000,C 90.000,E1 124.612} C_DIS
LIN {X -0.025,Y -510.872,Z 385.489,A 0.000,B 0.000,C 90.000,E1 123.992} C_DIS
LIN {X 0.131,Y -508.967,Z 385.484,A 0.000,B 0.000,C 90.000,E1 123.086} C_DIS
LIN {X 0.090,Y -507.525,Z 385.481,A 0.000,B 0.000,C 90.000,E1 122.498} C_DIS
LIN {X 0.203,Y -505.070,Z 385.476,A 0.000,B 0.000,C 90.000,E1 121.592} C_DIS
LIN {X 0.140,Y -503.258,Z 385.472,A 0.000,B 0.000,C 90.000,E1 121.003} C_DIS
LIN {X -0.063,Y -500.269,Z 385.467,A 0.000,B 0.000,C 90.000,E1 120.129} C_DIS
LIN {X 0.132,Y -496.933,Z 385.462,A 0.000,B 0.000,C 90.000,E1 119.205} C_DIS
LIN {X 0.081,Y -492.681,Z 385.457,A 0.000,B 0.000,C 90.000,E1 118.153} C_DIS
LIN {X -0.259,Y -488.121,Z 385.451,A 0.000,B 0.000,C 90.000,E1 117.129} C_DIS
LIN {X -0.005,Y -483.227,Z 385.445,A 0.000,B 0.000,C 90.000,E1 116.027} C_DIS
LIN {X -0.049,Y -476.643,Z 385.437,A 0.000,B 0.000,C 90.000,E1 114.643} C_DIS
LIN {X -0.165,Y -471.309,Z 385.431,A 0.000,B 0.000,C 90.000,E1 113.567} C_DIS
LIN {X -0.160,Y -464.240,Z 385.423,A 0.000,B 0.000,C 90.000,E1 112.153} C_DIS
LIN {X -0.098,Y -456.304,Z 385.414,A 0.000,B 0.000,C 90.000,E1 110.556} C_DIS
LIN {X -0.198,Y -455.618,Z 385.413,A 0.000,B 0.000,C 90.000,E1 110.429} C_DIS
LIN {X -0.238,Y -455.607,Z 385.413,A 0.000,B 0.000,C 90.000,E1 110.429} C_DIS
LIN {X 0.141,Y -457.000,Z 385.411,A 0.000,B 0.000,C 90.000,E1 109.885} C_DIS
LIN {X -0.050,Y -458.255,Z 385.407,A 0.000,B 0.000,C 90.000,E1 109.268} C_DIS
LIN {X 0.146,Y -466.418,Z 385.386,A 0.000,B 0.000,C 90.000,E1 105.426} C_DIS
LIN {X -0.129,Y -467.925,Z 385.382,A 0.000,B 0.000,C 90.000,E1 104.828} C_DIS
LIN {X -0.016,Y -475.501,Z 385.358,A 0.000,B 0.000,C 90.000,E1 100.423} C_DIS
LIN {X -0.264,Y -476.141,Z 385.356,A 0.000,B 0.000,C 90.000,E1 100.141} C_DIS
LIN {X 0.019,Y -482.054,Z 385.330,A 0.000,B 0.000,C 90.000,E1 95.454} C_DIS
LIN {X -0.190,Y -485.484,Z 385.305,A 0.000,B 0.000,C 90.000,E1 90.859} C_DIS
LIN {X -0.158,Y -486.386,Z 385.281,A 0.000,B 0.000,C 90.000,E1 86.560} C_DIS
LIN {X 0.152,Y -486.363,Z 385.279,A 0.000,B 0.000,C 90.000,E1 86.216} C_DIS
LIN {X 0.235,Y -484.689,Z 385.254,A 0.000,B 0.000,C 90.000,E1 81.602} C_DIS
LIN {X -0.016,Y -483.030,Z 385.245,A 0.000,B 0.000,C 90.000,E1 80.095} C_DIS
LIN {X 0.134,Y -480.621,Z 385.228,A 0.000,B 0.000,C 90.000,E1 76.992} C_DIS
LIN {X -0.008,Y -480.289,Z 385.226,A 0.000,B 0.000,C 90.000,E1 76.700} C_DIS
LIN {X -0.104,Y -474.112,Z 385.200,A 0.000,B 0.000,C 90.000,E1 72.054} C_DIS
LIN {X 0.200,Y -473.360,Z 385.198,A 0.000,B 0.000,C 90.000,E1 71.638} C_DIS
LIN {X 0.159,Y -473.392,Z 385.198,A 0.000,B 0.000,C 90.000,E1 71.638} C_DIS
LIN {X -0.100,Y -481.841,Z 385.192,A 0.000,B 0.000,C 90.000,E1 70.496} C_DIS
LIN {X -0.174,Y -491.564,Z 385.184,A 0.000,B 0.000,C 90.000,E1 69.135} C_DIS
LIN {X 0.156,Y -496.897,Z 385.180,A 0.000,B 0.000,C 90.000,E1 68.337} C_DIS
LIN {X -0.225,Y -502.863,Z 385.175,A 0.000,B 0.000,C 90.000,E1 67.486} C_DIS
LIN {X -0.230,Y -508.245,Z 385.170,A 0.000,B 0.000,C 90.000,E1 66.613} C_DIS
LIN {X -0.317,Y -510.948,Z 385.168,A 0.000,B 0.000,C 90.000,E1 66.177} C_DIS
LIN {X -0.064,Y -514.934,Z 385.163,A 0.000,B 0.000,C 90.000,E1 65.409} C_DIS
LIN {X 0.016,Y -518.621,Z 385.159,A 0.000,B 0.000,C 90.000,E1 64.665} C_DIS
LIN {X -0.119,Y -522.030,Z 385.155,A 0.000,B 0.000,C 90.000,E1 63.948} C_DIS
LIN {X 0.176,Y -524.508,Z 385.152,A 0.000,B 0.000,C 90.000,E1 63.332} C_DIS
LIN {X 0.252,Y -526.719,Z 385.149,A 0.000,B 0.000,C 90.000,E1 62.743} C_DIS
LIN {X -0.259,Y -530.736,Z 385.142,A 0.000,B 0.000,C 90.000,E1 61.641} C_DIS
LIN {X 0.004,Y -534.206,Z 385.136,A 0.000,B 0.000,C 90.000,E1 60.461} C_DIS
LIN {X -0.131,Y -536.650,Z 385.131,A 0.000,B 0.000,C 90.000,E1 59.616} C_DIS
LIN {X 0.029,Y -538.904,Z 385.126,A 0.000,B 0.000,C 90.000,E1 58.742} C_DIS
LIN {X 0.229,Y -541.638,Z 385.120,A 0.000,B 0.000,C 90.000,E1 57.582} C_DIS
LIN {X -0.280,Y -543.923,Z 385.114,A 0.000,B 0.000,C 90.000,E1 56.501} C_DIS
LIN {X 0.263,Y -545.401,Z 385.109,A 0.000,B 0.000,C 90.000,E1 55.595} C_DIS
LIN {X 0.063,Y -546.568,Z 385.104,A 0.000,B 0.000,C 90.000,E1 54.769} C_DIS
LIN {X 0.192,Y -547.421,Z 385.100,A 0.000,B 0.000,C 90.000,E1 53.909} C_DIS
LIN {X 0.003,Y -547.889,Z 385.095,A 0.000,B 0.000,C 90.000,E1 53.084} C_DIS
LIN {X -0.291,Y -548.159,Z 385.090,A 0.000,B 0.000,C 90.000,E1 52.271} C_DIS
LIN {X 0.195,Y -548.070,Z 385.086,A 0.000,B 0.000,C 90.000,E1 51.376} C_DIS
LIN {X -0.087,Y -547.718,Z 385.081,A 0.000,B 0.000,C 90.000,E1 50.561} C_DIS
LIN {X -0.332,Y -546.774,Z 385.075,A 0.000,B 0.000,C 90.000,E1 49.461} C_DIS
LIN {X 0.136,Y -545.847,Z 385.070,A 0.000,B 0.000,C 90.000,E1 48.566} C_DIS
LIN {X -0.195,Y -544.244,Z 385.064,A 0.000,B 0.000,C 90.000,E1 47.472} C_DIS
LIN {X 0.226,Y -541.733,Z 385.054,A 0.000,B 0.000,C 90.000,E1 45.729} C_DIS
LIN {X 0.183,Y -538.403,Z 385.042,A 0.000,B 0.000,C 90.000,E1 43.461} C_DIS
LIN {X 0.105,Y -536.117,Z 385.032,A 0.000,B 0.000,C 90.000,E1 41.757} C_DIS
LIN {X -0.034,Y -533.577,Z 385.021,A 0.000,B 0.000,C 90.000,E1 39.769} C_DIS
LIN {X 0.238,Y -530.996,Z 385.010,A 0.000,B 0.000,C 90.000,E1 37.729} C_DIS
LIN {X 0.165,Y -529.096,Z 385.002,A 0.000,B 0.000,C 90.000,E1 36.297} C_DIS
LIN {X 0.076,Y -527.565,Z 384.995,A 0.000,B 0.000,C 90.000,E1 35.152} C_DIS
LIN {X 0.027,Y -525.287,Z 384.986,A 0.000,B 0.000,C 90.000,E1 33.420} C_DIS
LIN {X 0.033,Y -522.646,Z 384.974,A 0.000,B 0.000,C 90.000,E1 31.386} C_DIS
LIN {X 0.148,Y -520.058,Z 384.963,A 0.000,B 0.000,C 90.000,E1 29.333} C_DIS
LIN {X 0.036,Y -517.963,Z 384.953,A 0.000,B 0.000,C 90.000,E1 27.590} C_DIS
LIN {X 0.009,Y -515.673,Z 384.942,A 0.000,B 0.000,C 90.000,E1 25.540} C_DIS
LIN {X -0.181,Y -513.272,Z 384.929,A 0.000,B 0.000,C 90.000,E1 23.206} C_DIS
LIN {X 0.292,Y -511.182,Z 384.916,A 0.000,B 0.000,C 90.000,E1 20.791} C_DIS
LIN {X 0.232,Y -509.641,Z 384.904,A 0.000,B 0.000,C 90.000,E1 18.725} C_DIS
LIN {X -0.120,Y -508.538,Z 384.894,A 0.000,B 0.000,C 90.000,E1 16.985} C_DIS
LIN {X -0.060,Y -507.471,Z 384.883,A 0.000,B 0.000,C 90.000,E1 14.898} C_DIS
LIN {X -0.163,Y -506.684,Z 384.871,A 0.000,B 0.000,C 90.000,E1 12.827} C_DIS
LIN {X -0.164,Y -506.190,Z 384.855,A 0.000,B 0.000,C 90.000,E1 9.849} C_DIS
LIN {X 0.207,Y -506.411,Z 384.840,A 0.000,B 0.000,C 90.000,E1 7.125} C_DIS
LIN {X 0.186,Y -507.734,Z 384.820,A 0.000,B 0.000,C 90.000,E1 3.555} C_DIS
LIN {X -0.218,Y -509.933,Z 384.803,A 0.000,B 0.000,C 90.000,E1 0.630} C_DIS
LIN {X -0.080,Y -514.339,Z 384.782,A 0.000,B 0.000,C 90.000,E1 356.846} C_DIS
LIN {X -0.125,Y -518.316,Z 384.768,A 0.000,B 0.000,C 90.000,E1 354.204} C_DIS
LIN {X 0.119,Y -522.478,Z 384.755,A 0.000,B 0.000,C 90.000,E1 351.837} C_DIS
LIN {X 0.277,Y -530.611,Z 384.734,A 0.000,B 0.000,C 90.000,E1 348.049} C_DIS
LIN {X -0.229,Y -537.309,Z 384.719,A 0.000,B 0.000,C 90.000,E1 345.519} C_DIS
LIN {X -0.030,Y -542.834,Z 384.708,A 0.000,B 0.000,C 90.000,E1 343.504} C_DIS
LIN {X -0.183,Y -545.250,Z 384.704,A 0.000,B 0.000,C 90.000,E1 342.670} C_DIS
LIN {X 0.184,Y -549.272,Z 384.696,A 0.000,B 0.000,C 90.000,E1 341.221} C_DIS
LIN {X -0.136,Y -554.191,Z 384.686,A 0.000,B 0.000,C 90.000,E1 339.571} C_DIS
LIN {X 0.073,Y -558.330,Z 384.679,A 0.000,B 0.000,C 90.000,E1 338.156} C_DIS
LIN {X 0.041,Y -561.604,Z 384.673,A 0.000,B 0.000,C 90.000,E1 337.050} C_DIS
LIN {X -0.106,Y -566.623,Z 384.663,A 0.000,B 0.000,C 90.000,E1 335.409} C_DIS
LIN {X -0.145,Y -571.698,Z 384.654,A 0.000,B 0.000,C 90.000,E1 333.768} C_DIS
LIN {X -0.005,Y -579.612,Z 384.641,A 0.000,B 0.000,C 90.000,E1 331.307} C_DIS
LIN {X -0.014,Y -586.863,Z 384.629,A 0.000,B 0.000,C 90.000,E1 329.154} C_DIS
LIN {X 0.293,Y -591.325,Z 384.621,A 0.000,B 0.000,C 90.000,E1 327.788} C_DIS
LIN {X -0.022,Y -597.623,Z 384.611,A 0.000,B 0.000,C 90.000,E1 325.960} C_DIS
LIN {X -0.009,Y -604.129,Z 384.601,A 0.000,B 0.000,C 90.000,E1 324.116} C_DIS
LIN {X 0.168,Y -610.694,Z 384.591,A 0.000,B 0.000,C 90.000,E1 322.271} C_DIS
LIN {X 0.089,Y -616.448,Z 384.582,A 0.000,B 0.000,C 90.000,E1 320.723} C_DIS
LIN {X -0.193,Y -621.316,Z 384.575,A 0.000,B 0.000,C 90.000,E1 319.461} C_DIS
LIN {X 0.206,Y -627.872,Z 384.565,A 0.000,B 0.000,C 90.000,E1 317.634} C_DIS
LIN {X 0.170,Y -631.542,Z 384.559,A 0.000,B 0.000,C 90.000,E1 316.620} C_DIS
LIN {X -0.275,Y -635.168,Z 384.554,A 0.000,B 0.000,C 90.000,E1 315.648} C_DIS
LIN {X 0.140,Y -639.743,Z 384.547,A 0.000,B 0.000,C 90.000,E1 314.352} C_DIS
LIN {X -0.201,Y -643.466,Z 384.541,A 0.000,B 0.000,C 90.000,E1 313.380} C_DIS
LIN {X -0.097,Y -648.118,Z 384.534,A 0.000,B 0.000,C 90.000,E1 312.123} C_DIS
LIN {X 0.086,Y -653.612,Z 384.526,A 0.000,B 0.000,C 90.000,E1 310.620} C_DIS
LIN {X -0.073,Y -659.735,Z 384.516,A 0.000,B 0.000,C 90.000,E1 308.910} C_DIS
LIN {X -0.074,Y -664.616,Z 384.508,A 0.000,B 0.000,C 90.000,E1 307.443} C_DIS
LIN {X 0.033,Y -668.531,Z 384.501,A 0.000,B 0.000,C 90.000,E1 306.217} C_DIS
LIN {X 0.222,Y -671.497,Z 384.496,A 0.000,B 0.000,C 90.000,E1 305.231} C_DIS
LIN {X 0.196,Y -675.757,Z 384.488,A 0.000,B 0.000,C 90.000,E1 303.785} C_DIS
LIN {X 0.106,Y -678.543,Z 384.482,A 0.000,B 0.000,C 90.000,E1 302.832} C_DIS
LIN {X 0.050,Y -681.118,Z 384.477,A 0.000,B 0.000,C 90.000,E1 301.878} C_DIS
LIN {X -0.177,Y -683.014,Z 384.473,A 0.000,B 0.000,C 90.000,E1 301.180} C_DIS
LIN {X 0.225,Y -684.322,Z 384.471,A 0.000,B 0.000,C 90.000,E1 300.669} C_DIS
LIN {X -0.114,Y -686.447,Z 384.465,A 0.000,B 0.000,C 90.000,E1 299.745} C_DIS
LIN {X -0.050,Y -687.770,Z 384.461,A 0.000,B 0.000,C 90.000,E1 299.027} C_DIS
LIN {X -0.118,Y -689.407,Z 384.455,A 0.000,B 0.000,C 90.000,E1 297.847} C_DIS
LIN {X -0.030,Y -690.044,Z 384.451,A 0.000,B 0.000,C 90.000,E1 297.129} C_DIS
LIN {X 0.061,Y -690.512,Z 384.447,A 0.000,B 0.000,C 90.000,E1 296.411} C_DIS
LIN {X -0.009,Y -690.506,Z 384.445,A 0.000,B 0.000,C 90.000,E1 296.181} C_DIS
LIN {X 0.231,Y -690.742,Z 384.444,A 0.000,B 0.000,C 90.000,E1 295.924} C_DIS
LIN {X 0.322,Y -690.940,Z 384.440,A 0.000,B 0.000,C 90.000,E1 295.207} C_DIS
LIN {X 0.068,Y -690.775,Z 384.435,A 0.000,B 0.000,C 90.000,E1 294.283} C_DIS
LIN {X -0.090,Y -690.591,Z 384.432,A 0.000,B 0.000,C 90.000,E1 293.823} C_DIS
LIN {X 0.334,Y -689.948,Z 384.428,A 0.000,B 0.000,C 90.000,E1 293.078} C_DIS
LIN {X 0.116,Y -689.048,Z 384.424,A 0.000,B 0.000,C 90.000,E1 292.386} C_DIS
LIN {X 0.301,Y -688.350,Z 384.422,A 0.000,B 0.000,C 90.000,E1 291.897} C_DIS
LIN {X -0.190,Y -687.236,Z 384.418,A 0.000,B 0.000,C 90.000,E1 291.227} C_DIS
LIN {X 0.198,Y -686.112,Z 384.414,A 0.000,B 0.000,C 90.000,E1 290.482} C_DIS
LIN {X -0.151,Y -683.884,Z 384.407,A 0.000,B 0.000,C 90.000,E1 289.322} C_DIS
LIN {X -0.107,Y -681.576,Z 384.401,A 0.000,B 0.000,C 90.000,E1 288.127} C_DIS
LIN {X 0.112,Y -679.235,Z 384.394,A 0.000,B 0.000,C 90.000,E1 286.913} C_DIS
LIN {X -0.062,Y -675.369,Z 384.383,A 0.000,B 0.000,C 90.000,E1 285.009} C_DIS
LIN {X -0.108,Y -669.856,Z 384.367,A 0.000,B 0.000,C 90.000,E1 282.119} C_DIS
LIN {X -0.028,Y -667.520,Z 384.359,A 0.000,B 0.000,C 90.000,E1 280.658} C_DIS
LIN {X 0.166,Y -664.523,Z 384.347,A 0.000,B 0.000,C 90.000,E1 278.454} C_DIS
LIN {X -0.307,Y -661.662,Z 384.331,A 0.000,B 0.000,C 90.000,E1 275.568} C_DIS
LIN {X 0.020,Y -660.236,Z 384.317,A 0.000,B 0.000,C 90.000,E1 273.094} C_DIS
LIN {X 0.193,Y -659.680,Z 384.304,A 0.000,B 0.000,C 90.000,E1 270.630} C_DIS
LIN {X -0.239,Y -659.565,Z 384.295,A 0.000,B 0.000,C 90.000,E1 269.198} C_DIS
LIN {X -0.313,Y -659.576,Z 384.290,A 0.000,B 0.000,C 90.000,E1 268.224} C_DIS
LIN {X 0.241,Y -659.666,Z 384.279,A 0.000,B 0.000,C 90.000,E1 266.216} C_DIS
LIN {X 0.187,Y -659.595,Z 384.274,A 0.000,B 0.000,C 90.000,E1 265.241} C_DIS
LIN {X -0.272,Y -659.435,Z 384.270,A 0.000,B 0.000,C 90.000,E1 264.546} C_DIS
LIN {X -0.007,Y -659.278,Z 384.267,A 0.000,B 0.000,C 90.000,E1 264.033} C_DIS
LIN {X -0.007,Y -658.704,Z 384.261,A 0.000,B 0.000,C 90.000,E1 263.053} C_DIS
LIN {X -0.138,Y -657.652,Z 384.255,A 0.000,B 0.000,C 90.000,E1 261.837} C_DIS
LIN {X 0.056,Y -656.493,Z 384.251,A 0.000,B 0.000,C 90.000,E1 261.084} C_DIS
LIN {X -0.004,Y -654.309,Z 384.244,A 0.000,B 0.000,C 90.000,E1 259.859} C_DIS
LIN {X 0.154,Y -652.803,Z 384.240,A 0.000,B 0.000,C 90.000,E1 259.106} C_DIS
LIN {X 0.030,Y -652.431,Z 384.238,A 0.000,B 0.000,C 90.000,E1 258.870} C_DIS
LIN {X 0.160,Y -650.959,Z 384.234,A 0.000,B 0.000,C 90.000,E1 258.117} C_DIS
LIN {X 0.140,Y -648.270,Z 384.227,A 0.000,B 0.000,C 90.000,E1 256.881} C_DIS
LIN {X -0.130,Y -647.105,Z 384.224,A 0.000,B 0.000,C 90.000,E1 256.408} C_DIS
LIN {X -0.212,Y -643.797,Z 384.218,A 0.000,B 0.000,C 90.000,E1 255.172} C_DIS
LIN {X -0.029,Y -640.850,Z 384.212,A 0.000,B 0.000,C 90.000,E1 254.157} C_DIS
LIN {X -0.052,Y -636.800,Z 384.205,A 0.000,B 0.000,C 90.000,E1 252.906} C_DIS
LIN {X 0.043,Y -632.365,Z 384.198,A 0.000,B 0.000,C 90.000,E1 251.638} C_DIS
LIN {X 0.264,Y -629.579,Z 384.194,A 0.000,B 0.000,C 90.000,E1 250.859} C_DIS
LIN {X -0.143,Y -624.664,Z 384.187,A 0.000,B 0.000,C 90.000,E1 249.625} C_DIS
LIN {X -0.034,Y -619.592,Z 384.180,A 0.000,B 0.000,C 90.000,E1 248.337} C_DIS
LIN {X -0.047,Y -613.236,Z 384.171,A 0.000,B 0.000,C 90.000,E1 246.794} C_DIS
LIN {X 0.042,Y -606.682,Z 384.162,A 0.000,B 0.000,C 90.000,E1 245.229} C_DIS
LIN {X 0.248,Y -600.050,Z 384.154,A 0.000,B 0.000,C 90.000,E1 243.640} C_DIS
LIN {X -0.132,Y -594.479,Z 384.146,A 0.000,B 0.000,C 90.000,E1 242.359} C_DIS
LIN {X 0.188,Y -589.002,Z 384.139,A 0.000,B 0.000,C 90.000,E1 241.001} C_DIS
LIN {X 0.085,Y -580.502,Z 384.127,A 0.000,B 0.000,C 90.000,E1 238.869} C_DIS
LIN {X 0.194,Y -571.503,Z 384.114,A 0.000,B 0.000,C 90.000,E1 236.421} C_DIS
LIN {X -0.132,Y -563.149,Z 384.100,A 0.000,B 0.000,C 90.000,E1 233.989} C_DIS
LIN {X 0.278,Y -559.474,Z 384.094,A 0.000,B 0.000,C 90.000,E1 232.844} C_DIS
LIN {X 0.193,Y -555.705,Z 384.088,A 0.000,B 0.000,C 90.000,E1 231.743} C_DIS
LIN {X 0.121,Y -550.894,Z 384.080,A 0.000,B 0.000,C 90.000,E1 230.356} C_DIS
LIN {X -0.030,Y -544.332,Z 384.069,A 0.000,B 0.000,C 90.000,E1 228.405} C_DIS
LIN {X -0.016,Y -537.986,Z 384.058,A 0.000,B 0.000,C 90.000,E1 226.419} C_DIS
LIN {X 0.253,Y -532.593,Z 384.048,A 0.000,B 0.000,C 90.000,E1 224.676} C_DIS
LIN {X 0.108,Y -529.081,Z 384.042,A 0.000,B 0.000,C 90.000,E1 223.542} C_DIS
LIN {X -0.182,Y -523.866,Z 384.032,A 0.000,B 0.000,C 90.000,E1 221.838} C_DIS
LIN {X 0.086,Y -517.958,Z 384.021,A 0.000,B 0.000,C 90.000,E1 219.769} C_DIS
LIN {X -0.065,Y -512.283,Z 384.010,A 0.000,B 0.000,C 90.000,E1 217.729} C_DIS
LIN {X -0.053,Y -506.043,Z 383.996,A 0.000,B 0.000,C 90.000,E1 215.358} C_DIS
LIN {X -0.156,Y -501.581,Z 383.987,A 0.000,B 0.000,C 90.000,E1 213.579} C_DIS
